(* IEC 61131-3 sources: RL_MAR/experiments/results/ablation/RL_MAR_DeepSeek-V3.2_full, 94 files *)

(* ---- hard_92.st ---- *)
TYPE
    BreakerState : STRUCT
        Opened : BOOL;
        Closed : BOOL;
    END_STRUCT;

    BreakerControl : STRUCT
        Trip : BOOL;
        Close : BOOL;
    END_STRUCT;

    BreakerData : STRUCT
        Control : BreakerControl;
        State : BreakerState;
    END_STRUCT;

    PointData : STRUCT
        Value : INT;
    END_STRUCT;
END_TYPE;

FUNCTION_BLOCK FB_BreakerControlSystem
VAR_INPUT
    B10_1_Trip : BOOL;
    B10_1_Close : BOOL;
    B10_2_Trip : BOOL;
    B10_2_Close : BOOL;
    B10_12_Trip : BOOL;
    B10_12_Close : BOOL;
    B54_Trip : BOOL;
    B54_Close : BOOL;
    B55_Trip : BOOL;
    B55_Close : BOOL;
    B56_Trip : BOOL;
    B56_Close : BOOL;
    B57_Trip : BOOL;
    B57_Close : BOOL;
END_VAR

VAR_OUTPUT
    Point_1a : INT;
    Point_2a : INT;
    Point_3a : INT;
    Point_4a : INT;
    B10_1_Opened : BOOL;
    B10_1_Closed : BOOL;
    B10_2_Opened : BOOL;
    B10_2_Closed : BOOL;
    B10_12_Opened : BOOL;
    B10_12_Closed : BOOL;
    B54_Opened : BOOL;
    B54_Closed : BOOL;
    B55_Opened : BOOL;
    B55_Closed : BOOL;
    B56_Opened : BOOL;
    B56_Closed : BOOL;
    B57_Opened : BOOL;
    B57_Closed : BOOL;
END_VAR

VAR
    SEL86_OUT : INT;
    MOVE89_OUT : INT;
    SEL66_OUT : INT;
    MOVE69_OUT : INT;
    SEL96_OUT : INT;
    MOVE99_OUT : INT;
    SEL106_OUT : INT;
    MOVE109_OUT : INT;
END_VAR

(* Breaker State Management *)
IF B10_1_Close = TRUE THEN
    B10_1_Closed := TRUE;
    B10_1_Opened := FALSE;
ELSIF B10_1_Trip = TRUE THEN
    B10_1_Closed := FALSE;
    B10_1_Opened := TRUE;
END_IF;

IF B10_2_Close = TRUE THEN
    B10_2_Closed := TRUE;
    B10_2_Opened := FALSE;
ELSIF B10_2_Trip = TRUE THEN
    B10_2_Closed := FALSE;
    B10_2_Opened := TRUE;
END_IF;

IF B10_12_Close = TRUE THEN
    B10_12_Closed := TRUE;
    B10_12_Opened := FALSE;
ELSIF B10_12_Trip = TRUE THEN
    B10_12_Closed := FALSE;
    B10_12_Opened := TRUE;
END_IF;

IF B54_Close = TRUE THEN
    B54_Closed := TRUE;
    B54_Opened := FALSE;
ELSIF B54_Trip = TRUE THEN
    B54_Closed := FALSE;
    B54_Opened := TRUE;
END_IF;

IF B55_Close = TRUE THEN
    B55_Closed := TRUE;
    B55_Opened := FALSE;
ELSIF B55_Trip = TRUE THEN
    B55_Closed := FALSE;
    B55_Opened := TRUE;
END_IF;

IF B56_Close = TRUE THEN
    B56_Closed := TRUE;
    B56_Opened := FALSE;
ELSIF B56_Trip = TRUE THEN
    B56_Closed := FALSE;
    B56_Opened := TRUE;
END_IF;

IF B57_Close = TRUE THEN
    B57_Closed := TRUE;
    B57_Opened := FALSE;
ELSIF B57_Trip = TRUE THEN
    B57_Closed := FALSE;
    B57_Opened := TRUE;
END_IF;

(* Point Calculations *)
IF (B54_Closed = TRUE) AND (((B10_12_Closed = TRUE) AND (B10_1_Closed = TRUE)) OR (B10_2_Closed = TRUE)) THEN
    Point_1a := 0;
ELSE
    Point_1a := 138;
END_IF;

IF (B55_Closed = TRUE) AND (((B10_12_Closed = TRUE) AND (B10_1_Closed = TRUE)) OR (B10_2_Closed = TRUE)) THEN
    Point_2a := 0;
ELSE
    Point_2a := 138;
END_IF;

IF (B56_Closed = TRUE) AND (((B10_12_Closed = TRUE) AND (B10_2_Closed = TRUE)) OR (B10_1_Closed = TRUE)) THEN
    Point_3a := 0;
ELSE
    Point_3a := 138;
END_IF;

IF (B57_Closed = TRUE) AND (((B10_12_Closed = TRUE) AND (B10_2_Closed = TRUE)) OR (B10_1_Closed = TRUE)) THEN
    Point_4a := 0;
ELSE
    Point_4a := 138;
END_IF;

END_FUNCTION_BLOCK;

(* ---- hard_93.st ---- *)
FUNCTION_BLOCK FB_CircuitControl
VAR_INPUT
    Reset_All_CB : BOOL;
    Current_Fault_on_TRSF1 : INT;
    Current_Fault_on_66BUS1 : INT;
END_VAR

VAR_OUTPUT
    Short_Circuit_TRSF1 : BOOL;
    Short_Circuit_66BUS : BOOL;
    Open_CB1_66KV : BOOL;
    Open_CB2_66KV : BOOL;
    Open_CB_TRSF1 : BOOL;
    Open_CB2_22KV : BOOL;
END_VAR

VAR
    Threshold500 : INT := 500;
    Prev_Open_CB2_22KV : BOOL;
    Prev_Open_CB1_66KV : BOOL;
    Prev_Open_CB_TRSF1 : BOOL;
    Temp_Open_CB2_22KV : BOOL;
    Temp_Open_CB1_66KV : BOOL;
    Temp_Open_CB_TRSF1 : BOOL;
END_VAR

(* Short circuit detection *)
Short_Circuit_66BUS := Current_Fault_on_66BUS1 > Threshold500;
Short_Circuit_TRSF1 := Current_Fault_on_TRSF1 > Threshold500;

(* Set Open_CB2_66KV to TRUE as specified *)
Open_CB2_66KV := TRUE;

(* Reset logic - when Reset_All_CB is TRUE, close all breakers and reset previous states *)
IF Reset_All_CB THEN
    Open_CB2_22KV := FALSE;
    Open_CB1_66KV := FALSE;
    Open_CB_TRSF1 := FALSE;
    Prev_Open_CB2_22KV := FALSE;
    Prev_Open_CB1_66KV := FALSE;
    Prev_Open_CB_TRSF1 := FALSE;
ELSE
    (* First calculation of breaker states *)
    Temp_Open_CB2_22KV := (NOT Prev_Open_CB2_22KV) AND ((Open_CB1_66KV AND Open_CB_TRSF1) OR Short_Circuit_66BUS);
    Temp_Open_CB1_66KV := (NOT Temp_Open_CB2_22KV) AND ((Prev_Open_CB1_66KV AND Open_CB_TRSF1) OR Short_Circuit_66BUS);
    Temp_Open_CB_TRSF1 := (NOT Temp_Open_CB2_22KV) AND ((Open_CB1_66KV AND Prev_Open_CB_TRSF1) OR Short_Circuit_66BUS);

    (* Update with Open_CB2_66KV and Short_Circuit_TRSF1 conditions *)
    Temp_Open_CB2_22KV := (NOT Prev_Open_CB2_22KV) AND ((Open_CB2_66KV AND Open_CB1_66KV AND Open_CB_TRSF1) OR Short_Circuit_TRSF1);
    Temp_Open_CB1_66KV := (NOT Temp_Open_CB2_22KV) AND ((Open_CB2_66KV AND Prev_Open_CB1_66KV AND Open_CB_TRSF1) OR Short_Circuit_TRSF1);
    Temp_Open_CB_TRSF1 := (NOT Temp_Open_CB2_22KV) AND ((Open_CB2_66KV AND Open_CB1_66KV AND Prev_Open_CB_TRSF1) OR Short_Circuit_TRSF1);

    (* Assign final values to outputs *)
    Open_CB2_22KV := Temp_Open_CB2_22KV;
    Open_CB1_66KV := Temp_Open_CB1_66KV;
    Open_CB_TRSF1 := Temp_Open_CB_TRSF1;

    (* Store current states as previous for next scan *)
    Prev_Open_CB2_22KV := Open_CB2_22KV;
    Prev_Open_CB1_66KV := Open_CB1_66KV;
    Prev_Open_CB_TRSF1 := Open_CB_TRSF1;
END_IF;

END_FUNCTION_BLOCK;

(* ---- hard_94.st ---- *)
FUNCTION_BLOCK FB_AdvancedCircuitBreakerControl
    VAR_INPUT
        S_AL1_P_B1 : BOOL;
        S_AL1_P_B2 : BOOL;
        S_AL1_MCB : BOOL;
        MCB_BUSY : BOOL;
        MCB_ERROR : BOOL;
        S_AL1_MCBR : BOOL;
        MCBR_BUSY : BOOL;
        MCBR_ERROR : BOOL;
        S_AL1_P_B3 : BOOL;
        S_AL1_MCB2 : BOOL;
        S_AL1_MCBR2 : BOOL;
    END_VAR

    VAR_OUTPUT
        E_AL1_B1 : BOOL;
        PUWS_AL1_B1_PLUS : BOOL;
        PUWS_AL1_B1_RIGHT : BOOL;
        PAS_AL1_PLUS : BOOL;
        PAS_AL1_TURN : BOOL;
    END_VAR

    VAR
        PPAL1 : BOOL := 1;
        PP0 : BOOL := 1;
        PP1 : BOOL := 0;
        PP2 : BOOL := 0;
        PP3 : BOOL := 0;
        PP4 : BOOL := 0;
        MCB : BOOL := 1;
        PP5 : BOOL := 0;
        PP7 : BOOL := 0;
        PPL3 : BOOL := 0;
        PPL4 : BOOL := 0;
        MCBR : BOOL := 1;
        PPL5 : BOOL := 0;
        PPL7 : BOOL := 0;
        STABLE : BOOL := 0;
        MCB_CONTROL : BOOL;
    END_VAR

    STABLE := 0;
    WHILE (STABLE = 0) DO
        STABLE := 1;
        IF PP0 AND (NOT MCB_CONTROL) AND (NOT PP1) THEN
            PP0 := 0;
            PP1 := 1;
            STABLE := 0;
        END_IF;
        IF PP1 AND S_AL1_P_B1 AND (NOT PP2) THEN
            PP1 := 0;
            PP2 := 1;
            STABLE := 0;
        END_IF;
        IF PP2 AND S_AL1_P_B2 AND (NOT MCB_CONTROL) AND (NOT PP3) THEN
            PP2 := 0;
            PP3 := 1;
            STABLE := 0;
        END_IF;
        IF PP3 AND S_AL1_MCB AND (NOT PP4) AND (NOT PP1) THEN
            PP3 := 0;
            PP4 := 1;
            PP1 := 1;
            STABLE := 0;
        END_IF;
        IF PP4 AND MCB AND MCB_BUSY AND (NOT PP5) THEN
            PP4 := 0;
            MCB := 0;
            PP5 := 1;
            STABLE := 0;
        END_IF;
        IF PP5 AND S_AL1_MCB2 AND (NOT PP7) AND (NOT MCB) THEN
            PP5 := 0;
            PP7 := 1;
            MCB := 1;
            STABLE := 0;
        END_IF;
        IF PP7 AND S_AL1_P_B3 THEN
            PP7 := 0;
            STABLE := 0;
        END_IF;
        IF PP2 AND S_AL1_P_B2 AND MCB_CONTROL AND (NOT PPL3) AND (NOT PP1) THEN
            PP2 := 0;
            PPL3 := 1;
            PP1 := 1;
            STABLE := 0;
        END_IF;
        IF PPL3 AND S_AL1_MCBR AND (NOT PPL4) THEN
            PPL3 := 0;
            PPL4 := 1;
            STABLE := 0;
        END_IF;
        IF PPL4 AND MCBR AND MCBR_BUSY AND (NOT PPL5) THEN
            PPL4 := 0;
            MCBR := 0;
            PPL5 := 1;
            STABLE := 0;
        END_IF;
        IF PPL5 AND S_AL1_MCBR2 AND (NOT PPL7) AND (NOT MCBR) THEN
            PPL5 := 0;
            PPL7 := 1;
            MCBR := 1;
            STABLE := 0;
        END_IF;
        IF PPL7 AND S_AL1_P_B3 THEN
            PPL7 := 0;
            STABLE := 0;
        END_IF;
    END_WHILE;

    IF PP0 OR PP1 THEN
        E_AL1_B1 := 1;
    END_IF;
    IF PP3 THEN
        MCB_CONTROL := 1;
    END_IF;
    IF PPL3 OR PPL4 THEN
        PAS_AL1_PLUS := 1;
        PAS_AL1_TURN := 1;
    END_IF;
    IF PPAL1 OR PP2 THEN
        PUWS_AL1_B1_PLUS := 1;
    END_IF;
    IF PP2 OR PP3 OR PPL3 THEN
        E_AL1_B1 := 0;
    END_IF;
    IF PP0 OR PP3 THEN
        MCB_CONTROL := 0;
    END_IF;
    IF PP0 OR PP3 OR PP4 THEN
        PAS_AL1_PLUS := 0;
        PAS_AL1_TURN := 0;
    END_IF;
    IF PPAL1 OR PP2 THEN
        PUWS_AL1_B1_RIGHT := 0;
    END_IF;
END_FUNCTION_BLOCK;

(* ---- hf_1.st ---- *)
FUNCTION_BLOCK StackMin
VAR_INPUT
    push : BOOL;
    pop : BOOL;
    reset : BOOL;
END_VAR

VAR_OUTPUT
    error : BOOL;
    status : WORD;
END_VAR

VAR_IN_OUT
    item : INT;
    stack : ARRAY[0..3] OF INT;
END_VAR

VAR
    top : INT := -1;
    i : INT;
    j : INT;
    minIndex : INT;
    minValue : INT;
END_VAR

IF reset THEN
    top := -1;
    error := FALSE;
    status := 16#0000;
ELSIF push THEN
    IF top >= 3 THEN
        error := TRUE;
        status := 16#8A04;
    ELSE
        top := top + 1;
        stack[top] := item;
        error := FALSE;
        status := 16#0000;
    END_IF;
ELSIF pop THEN
    IF top < 0 THEN
        error := TRUE;
        status := 16#8A05;
    ELSE
        minIndex := 0;
        minValue := stack[0];
        i := 1;
        WHILE i <= top DO
            IF stack[i] < minValue THEN
                minValue := stack[i];
                minIndex := i;
            END_IF;
            i := i + 1;
        END_WHILE;
        item := minValue;
        j := minIndex;
        WHILE j < top DO
            stack[j] := stack[j + 1];
            j := j + 1;
        END_WHILE;
        top := top - 1;
        error := FALSE;
        status := 16#0000;
    END_IF;
ELSE
    error := FALSE;
    status := 16#0000;
END_IF;

END_FUNCTION_BLOCK;

(* ---- hf_10.st ---- *)
FUNCTION_BLOCK FloatingAverage
VAR_INPUT
    cyclicExecution : BOOL;
    trigger : BOOL;
    value : REAL;
    windowSize : INT;
    reset : BOOL;
END_VAR

VAR_OUTPUT
    average : REAL;
    windowSizeReached : BOOL;
    error : BOOL;
    status : WORD;
END_VAR

VAR
    dataBuffer : ARRAY[1..100] OF REAL;
    bufferIndex : INT := 1;
    sum : REAL := 0.0;
    elementCount : INT := 0;
    triggerPrev : BOOL := FALSE;
    i : INT;
END_VAR

IF reset THEN
    sum := 0.0;
    average := 0.0;
    elementCount := 0;
    bufferIndex := 1;
    windowSizeReached := FALSE;
    error := FALSE;
    status := 16#0000;

    FOR i := 1 TO 100 DO
        dataBuffer[i] := 0.0;
    END_FOR;
ELSE
    IF (windowSize < 1) OR (windowSize > 100) THEN
        error := TRUE;
        status := 16#8200;
        average := 0.0;
        windowSizeReached := FALSE;
    ELSE
        error := FALSE;
        status := 16#0000;

        IF cyclicExecution THEN
            sum := sum - dataBuffer[bufferIndex];
            dataBuffer[bufferIndex] := value;
            sum := sum + value;

            bufferIndex := bufferIndex + 1;
            IF bufferIndex > windowSize THEN
                bufferIndex := 1;
            END_IF;

            IF elementCount < windowSize THEN
                elementCount := elementCount + 1;
            END_IF;
        ELSE
            IF trigger AND NOT triggerPrev THEN
                sum := sum - dataBuffer[bufferIndex];
                dataBuffer[bufferIndex] := value;
                sum := sum + value;

                bufferIndex := bufferIndex + 1;
                IF bufferIndex > windowSize THEN
                    bufferIndex := 1;
                END_IF;

                IF elementCount < windowSize THEN
                    elementCount := elementCount + 1;
                END_IF;
            END_IF;
            triggerPrev := trigger;
        END_IF;

        IF elementCount >= windowSize THEN
            windowSizeReached := TRUE;
            average := sum / INT_TO_REAL(windowSize);
        ELSE
            windowSizeReached := FALSE;
            IF elementCount > 0 THEN
                average := sum / INT_TO_REAL(elementCount);
            ELSE
                average := 0.0;
            END_IF;
        END_IF;
    END_IF;
END_IF;
END_FUNCTION_BLOCK

(* ---- hf_11.st ---- *)
FUNCTION_BLOCK FB_BottleProcessing
VAR_INPUT
    bottleSensor : BOOL;
    cleaningConfirmButton : BOOL;
    fillingConfirmButton : BOOL;
    cappingConfirmButton : BOOL;
    packingConfirmButton : BOOL;
    finishedButton : BOOL;
END_VAR

VAR_OUTPUT
    Pump_Motor : BOOL;
    Filling_Valve : BOOL;
    Capping_Machine : BOOL;
    Packing_Machine : BOOL;
    Completion_Light : BOOL;
END_VAR

VAR
    State : INT := 0;
END_VAR

CASE State OF
    0:
        Pump_Motor := FALSE;
        Filling_Valve := FALSE;
        Capping_Machine := FALSE;
        Packing_Machine := FALSE;
        Completion_Light := FALSE;

        IF bottleSensor THEN
            State := 1;
        END_IF;

    1:
        Pump_Motor := TRUE;
        Filling_Valve := FALSE;
        Capping_Machine := FALSE;
        Packing_Machine := FALSE;
        Completion_Light := FALSE;

        IF cleaningConfirmButton THEN
            State := 2;
        END_IF;

    2:
        Pump_Motor := FALSE;
        Filling_Valve := TRUE;
        Capping_Machine := FALSE;
        Packing_Machine := FALSE;
        Completion_Light := FALSE;

        IF fillingConfirmButton THEN
            State := 3;
        END_IF;

    3:
        Pump_Motor := FALSE;
        Filling_Valve := FALSE;
        Capping_Machine := TRUE;
        Packing_Machine := FALSE;
        Completion_Light := FALSE;

        IF cappingConfirmButton THEN
            State := 4;
        END_IF;

    4:
        Pump_Motor := FALSE;
        Filling_Valve := FALSE;
        Capping_Machine := FALSE;
        Packing_Machine := TRUE;
        Completion_Light := FALSE;

        IF packingConfirmButton THEN
            State := 5;
        END_IF;

    5:
        Pump_Motor := FALSE;
        Filling_Valve := FALSE;
        Capping_Machine := FALSE;
        Packing_Machine := FALSE;
        Completion_Light := TRUE;

        IF finishedButton THEN
            State := 0;
        END_IF;

    ELSE
        State := 0;
        Pump_Motor := FALSE;
        Filling_Valve := FALSE;
        Capping_Machine := FALSE;
        Packing_Machine := FALSE;
        Completion_Light := FALSE;
END_CASE;
END_FUNCTION_BLOCK

(* ---- hf_12.st ---- *)
FUNCTION_BLOCK MaterialMixing
VAR_INPUT
    estop : BOOL; (* Emergency Stop Signal, FALSE: Emergency stop triggered, TRUE: No emergency stop triggered *)
    opeMode : BOOL; (* Operation Mode, FALSE: Manual Operation Mode, TRUE: Automatic Operation Mode *)
    valveAStart : BOOL; (* Valve A Start Button *)
    valveBStart : BOOL; (* Valve B Start Button *)
    valveCStart : BOOL; (* Valve C Start Button *)
    valveDStart : BOOL; (* Valve D Start Button *)
    mixMotorStart : BOOL; (* Mixing Motor Start Button *)
    autoStart : BOOL; (* Automatic Start Button *)
    processMode : BOOL; (* Process Mode *)
    levelSensor : INT; (* Liquid Level Sensor, unit cm *)
    mixMotorComplete : BOOL; (* Mixing Complete Signal *)
END_VAR

VAR_OUTPUT
    valveARun : BOOL; (* Valve A Run Command *)
    valveBRun : BOOL; (* Valve B Run Command *)
    valveCRun : BOOL; (* Valve C Run Command *)
    valveDRun : BOOL; (* Valve D Run Command *)
    mixMotorRun : BOOL; (* Mixing Motor Run Command *)
END_VAR

VAR
    previousValveAStart : BOOL := FALSE;
    previousValveBStart : BOOL := FALSE;
    previousValveCStart : BOOL := FALSE;
    previousValveDStart : BOOL := FALSE;
    previousMixMotorStart : BOOL := FALSE;
    previousAutoStart : BOOL := FALSE;
END_VAR

(* Emergency Stop has highest priority - override all other logic *)
IF NOT estop THEN
    (* Automatic Operation Mode *)
    IF opeMode THEN
        (* Rising edge detection for autoStart button *)
        IF autoStart AND NOT previousAutoStart THEN
            valveARun := TRUE;
            valveBRun := FALSE;
            valveCRun := FALSE;
            valveDRun := FALSE;
            mixMotorRun := FALSE;
        END_IF;

        (* Automatic sequence logic *)
        IF valveARun AND (levelSensor >= 50) THEN
            valveARun := FALSE;
            valveBRun := TRUE;
        END_IF;

        IF valveBRun AND (levelSensor >= 80) THEN
            valveBRun := FALSE;
            IF processMode THEN
                valveCRun := TRUE;
            ELSE
                mixMotorRun := TRUE;
            END_IF;
        END_IF;

        IF valveCRun AND (levelSensor >= 100) THEN
            valveCRun := FALSE;
            mixMotorRun := TRUE;
        END_IF;

        IF mixMotorRun AND mixMotorComplete THEN
            mixMotorRun := FALSE;
            valveDRun := TRUE;
        END_IF;
    (* Manual Operation Mode *)
    ELSE
        (* Toggle logic with rising edge detection for manual buttons *)
        IF valveAStart AND NOT previousValveAStart THEN
            valveARun := NOT valveARun;
        END_IF;

        IF valveBStart AND NOT previousValveBStart THEN
            valveBRun := NOT valveBRun;
        END_IF;

        IF valveCStart AND NOT previousValveCStart THEN
            valveCRun := NOT valveCRun;
        END_IF;

        IF valveDStart AND NOT previousValveDStart THEN
            valveDRun := NOT valveDRun;
        END_IF;

        IF mixMotorStart AND NOT previousMixMotorStart THEN
            mixMotorRun := NOT mixMotorRun;
        END_IF;
    END_IF;
(* Emergency Stop active - force all outputs to FALSE *)
ELSE
    valveARun := FALSE;
    valveBRun := FALSE;
    valveCRun := FALSE;
    valveDRun := FALSE;
    mixMotorRun := FALSE;
END_IF;

(* Update previous state variables for edge detection *)
previousValveAStart := valveAStart;
previousValveBStart := valveBStart;
previousValveCStart := valveCStart;
previousValveDStart := valveDStart;
previousMixMotorStart := mixMotorStart;
previousAutoStart := autoStart;

END_FUNCTION_BLOCK;

(* ---- hf_13.st ---- *)
FUNCTION_BLOCK TON
VAR_INPUT
    IN : BOOL;
    PT : DINT;
    CYCLE_TIME : DINT;
END_VAR
VAR_OUTPUT
    Q : BOOL;
    ET : DINT;
END_VAR
VAR
    elapsedTimeInternal : DINT := 0;
    IN_PREV : BOOL := FALSE;
END_VAR

IF IN THEN
    IF NOT IN_PREV THEN
        elapsedTimeInternal := 0;
    END_IF;

    IF elapsedTimeInternal < PT THEN
        elapsedTimeInternal := elapsedTimeInternal + CYCLE_TIME;
        Q := FALSE;
    ELSE
        elapsedTimeInternal := PT;
        Q := TRUE;
    END_IF;

    ET := elapsedTimeInternal;
ELSE
    Q := FALSE;
    ET := 0;
    elapsedTimeInternal := 0;
END_IF;

IN_PREV := IN;
END_FUNCTION_BLOCK;

FUNCTION_BLOCK LightsControl
VAR_INPUT
    button1 : BOOL;
    button2 : BOOL;
    button3 : BOOL;
    CYCLE_TIME : DINT;
END_VAR
VAR_OUTPUT
    greenLight : BOOL;
    redLight : BOOL;
    yellowLight : BOOL;
END_VAR
VAR
    timerAuto : TON;
    timerGreen : TON;
    timerRed : TON;
    timerYellow : TON;
    currentState : INT := 0;
    autoRunTimer : BOOL;
END_VAR

IF NOT button1 THEN
    timerGreen(IN:=FALSE, PT:=1000, CYCLE_TIME:=CYCLE_TIME);
    timerRed(IN:=FALSE, PT:=1000, CYCLE_TIME:=CYCLE_TIME);
    timerYellow(IN:=FALSE, PT:=500, CYCLE_TIME:=CYCLE_TIME);

    IF NOT button2 AND NOT button3 THEN
        greenLight := FALSE;
        redLight := FALSE;
        yellowLight := FALSE;
    ELSIF button2 AND NOT button3 THEN
        greenLight := TRUE;
        timerRed(IN:=TRUE, PT:=1000, CYCLE_TIME:=CYCLE_TIME);
        redLight := timerRed.Q;
        yellowLight := FALSE;
    ELSIF NOT button2 AND button3 THEN
        redLight := TRUE;
        timerYellow(IN:=TRUE, PT:=500, CYCLE_TIME:=CYCLE_TIME);
        yellowLight := NOT timerYellow.Q;
        greenLight := FALSE;
    ELSIF button2 AND button3 THEN
        yellowLight := TRUE;
        timerGreen(IN:=TRUE, PT:=500, CYCLE_TIME:=CYCLE_TIME);
        greenLight := NOT timerGreen.Q;
        redLight := FALSE;
    END_IF;
ELSE
    autoRunTimer := TRUE;
    timerAuto(IN:=autoRunTimer, PT:=1000, CYCLE_TIME:=CYCLE_TIME);

    IF timerAuto.Q THEN
        currentState := currentState + 1;
        IF currentState > 2 THEN
            currentState := 0;
        END_IF;
        timerAuto(IN:=FALSE, PT:=1000, CYCLE_TIME:=CYCLE_TIME);
        timerAuto(IN:=TRUE, PT:=1000, CYCLE_TIME:=CYCLE_TIME);
    END_IF;

    CASE currentState OF
        0:
            greenLight := TRUE;
            redLight := FALSE;
            yellowLight := FALSE;
        1:
            greenLight := FALSE;
            redLight := TRUE;
            yellowLight := FALSE;
        2:
            greenLight := FALSE;
            redLight := FALSE;
            yellowLight := TRUE;
        ELSE
            currentState := 0;
            greenLight := TRUE;
            redLight := FALSE;
            yellowLight := FALSE;
    END_CASE;
END_IF;
END_FUNCTION_BLOCK;

(* ---- hf_14.st ---- *)
FUNCTION_BLOCK TruckGarage
VAR_INPUT
    enter_flag : BOOL;
    exit_flag : BOOL;
    VehicleNumber_in : INT;
END_VAR
VAR_OUTPUT
    truck_row : INT;
    truck_col : INT;
    truck_VehicleNumber : INT;
END_VAR
VAR_IN_OUT
    garage : ARRAY[1..3, 1..5] OF STRUCT
        Occupied : BOOL;
        VehicleNumber : INT;
    END_STRUCT;
END_VAR
VAR
    i : INT;
    j : INT;
    entry_found : BOOL;
    exit_found : BOOL;
END_VAR

// Initialize output
truck_row := 0;
truck_col := 0;
truck_VehicleNumber := 0;

// Entry logic
IF enter_flag THEN
    entry_found := FALSE;

    // Search from last row to first, last column to first
    FOR i := 3 TO 1 BY -1 DO
        FOR j := 5 TO 1 BY -1 DO
            IF NOT garage[i, j].Occupied AND NOT entry_found THEN
                // Allocate this space
                garage[i, j].Occupied := TRUE;
                garage[i, j].VehicleNumber := VehicleNumber_in;
                entry_found := TRUE;
            END_IF;
        END_FOR;
    END_FOR;
END_IF;

// Exit logic
IF exit_flag THEN
    exit_found := FALSE;

    // Search from first row to last, first column to last
    FOR i := 1 TO 3 DO
        FOR j := 1 TO 5 DO
            IF garage[i, j].Occupied AND (garage[i, j].VehicleNumber = VehicleNumber_in) AND NOT exit_found THEN
                // Release this space
                garage[i, j].Occupied := FALSE;
                garage[i, j].VehicleNumber := 0;

                // Set output information
                truck_row := i;
                truck_col := j;
                truck_VehicleNumber := VehicleNumber_in;
                exit_found := TRUE;
            END_IF;
        END_FOR;
    END_FOR;
END_IF;

END_FUNCTION_BLOCK

(* ---- hf_15.st ---- *)
FUNCTION_BLOCK FB_MergeBytes
VAR_INPUT
    byteArray : ARRAY[1..20] OF DINT; (* Byte array to be merged *)
END_VAR

VAR_OUTPUT
    dwordArray : ARRAY[1..10] OF DINT; (* Merged double word array *)
    mergeDwordNum : DINT; (* Actual number of merged double words *)
END_VAR

VAR
    i : DINT; (* Input byte index *)
    j : DINT; (* Byte counter within group (0-3) *)
    k : DINT; (* Output array index *)
    tempDword : DINT; (* Temporary storage for building double word *)
    currentByteValue : DINT; (* Temporary storage for current byte *)
END_VAR

VAR CONSTANT
    BYTE_ARRAY_SIZE : DINT := 20; (* Size of the input byte array *)
    DWORD_ARRAY_SIZE : DINT := 10; (* Size of the output DINT array *)
END_VAR

(* Initialize output count *)
mergeDwordNum := 0;

(* Clear output array *)
FOR k := 1 TO DWORD_ARRAY_SIZE DO
    dwordArray[k] := 0;
END_FOR;

(* Main merging loop *)
i := 1;
WHILE i <= BYTE_ARRAY_SIZE DO
    tempDword := 0;
    j := 0;

    (* Collect up to 4 bytes *)
    WHILE (j < 4) AND ((i + j) <= BYTE_ARRAY_SIZE) DO
        currentByteValue := byteArray[i + j];
        currentByteValue := currentByteValue AND 16#FF; (* Mask to keep only LSB *)
        tempDword := tempDword OR SHL(currentByteValue, 8 * j); (* Shift and combine *)
        j := j + 1;
    END_WHILE;

    (* Check if we have a complete group of 4 bytes *)
    IF j = 4 THEN
        k := mergeDwordNum + 1;

        (* Check if output array has space *)
        IF k <= DWORD_ARRAY_SIZE THEN
            dwordArray[k] := tempDword;
            mergeDwordNum := k;
        ELSE
            EXIT; (* Output array full *)
        END_IF;
    ELSE
        EXIT; (* Incomplete byte group *)
    END_IF;

    i := i + 4; (* Move to next group *)
END_WHILE;

END_FUNCTION_BLOCK;

(* ---- hf_16.st ---- *)
FUNCTION_BLOCK FB_LinearizeValue
VAR_INPUT
    InputValue : REAL; // Floating point input, raw measurement value
END_VAR

VAR_OUTPUT
    LinearizedValue : REAL; // Converted linear value
    Error : BOOL; // Error status indicator
    Status : WORD; // Status code
END_VAR

VAR
    // Internal constants for the piecewise linear segments
    RANGE1_IN_MIN : REAL := 1200.0;
    RANGE1_IN_MAX : REAL := 3600.0;
    RANGE1_OUT_MIN : REAL := 150.0;
    RANGE1_OUT_MAX : REAL := 240.0;

    RANGE2_IN_MIN : REAL := 3600.0;
    RANGE2_IN_MAX : REAL := 4800.0;
    RANGE2_OUT_MIN : REAL := 240.0;
    RANGE2_OUT_MAX : REAL := 560.0;

    RANGE3_IN_MIN : REAL := 4800.0;
    RANGE3_IN_MAX : REAL := 7000.0;
    RANGE3_OUT_MIN : REAL := 560.0;
    RANGE3_OUT_MAX : REAL := 720.0;

    // Status codes
    STATUS_SUCCESS : WORD := 16#0000;
    STATUS_OUT_OF_RANGE : WORD := 16#8001;
END_VAR

// Main execution logic
IF InputValue < RANGE1_IN_MIN THEN
    // Below minimum range
    LinearizedValue := RANGE1_OUT_MIN;
    Error := TRUE;
    Status := STATUS_OUT_OF_RANGE;
ELSIF InputValue >= RANGE1_IN_MIN AND InputValue <= RANGE1_IN_MAX THEN
    // Range 1: 1200 to 3600
    LinearizedValue := RANGE1_OUT_MIN + (InputValue - RANGE1_IN_MIN) *
                      (RANGE1_OUT_MAX - RANGE1_OUT_MIN) /
                      (RANGE1_IN_MAX - RANGE1_IN_MIN);
    Error := FALSE;
    Status := STATUS_SUCCESS;
ELSIF InputValue > RANGE1_IN_MAX AND InputValue <= RANGE2_IN_MAX THEN
    // Range 2: 3600 to 4800
    LinearizedValue := RANGE2_OUT_MIN + (InputValue - RANGE2_IN_MIN) *
                      (RANGE2_OUT_MAX - RANGE2_OUT_MIN) /
                      (RANGE2_IN_MAX - RANGE2_IN_MIN);
    Error := FALSE;
    Status := STATUS_SUCCESS;
ELSIF InputValue > RANGE2_IN_MAX AND InputValue <= RANGE3_IN_MAX THEN
    // Range 3: 4800 to 7000
    LinearizedValue := RANGE3_OUT_MIN + (InputValue - RANGE3_IN_MIN) *
                      (RANGE3_OUT_MAX - RANGE3_OUT_MIN) /
                      (RANGE3_IN_MAX - RANGE3_IN_MIN);
    Error := FALSE;
    Status := STATUS_SUCCESS;
ELSE
    // Above maximum range
    LinearizedValue := RANGE3_OUT_MAX;
    Error := TRUE;
    Status := STATUS_OUT_OF_RANGE;
END_IF;

END_FUNCTION_BLOCK

(* ---- hf_17.st ---- *)
FUNCTION_BLOCK FB_WarehouseManagement
VAR_INPUT
    requestIn : BOOL := FALSE;
    requestOut : BOOL := FALSE;
END_VAR

VAR_OUTPUT
    productNum : INT := 0;
    libFreeNum : INT := 9;
    error : BOOL := FALSE;
    status : WORD := 16#0000;
END_VAR

VAR_IN_OUT
    library : ARRAY[1..9] OF BOOL;
END_VAR

VAR
    i : INT;
    found : BOOL;
    initDone : BOOL := FALSE;
    errFull : WORD := 16#8001;
    errEmpty : WORD := 16#8002;
END_VAR

// Initialize library array on first execution
IF NOT initDone THEN
    i := 1;
    WHILE i <= 9 DO
        library[i] := FALSE;
        i := i + 1;
    END_WHILE;
    initDone := TRUE;
END_IF;

// Reset error status at start of each cycle
error := FALSE;
status := 16#0000;

// Handle storage request
IF requestIn THEN
    // Check if storage is full
    IF productNum >= 9 THEN
        error := TRUE;
        status := errFull;
    ELSE
        // Search for free position from highest to lowest index (9 to 1)
        found := FALSE;
        i := 9;
        WHILE i >= 1 AND NOT found DO
            IF NOT library[i] THEN
                library[i] := TRUE;
                productNum := productNum + 1;
                libFreeNum := libFreeNum - 1;
                found := TRUE;
            END_IF;
            i := i - 1;
        END_WHILE;

        // If no free position found despite productNum < 9, set error
        IF NOT found THEN
            error := TRUE;
            status := errFull;
        END_IF;
    END_IF;
END_IF;

// Handle retrieval request
IF requestOut THEN
    // Check if storage is empty
    IF productNum <= 0 THEN
        error := TRUE;
        status := errEmpty;
    ELSE
        // Search for occupied position from lowest to highest index (1 to 9)
        found := FALSE;
        i := 1;
        WHILE i <= 9 AND NOT found DO
            IF library[i] THEN
                library[i] := FALSE;
                productNum := productNum - 1;
                libFreeNum := libFreeNum + 1;
                found := TRUE;
            END_IF;
            i := i + 1;
        END_WHILE;

        // If no occupied position found despite productNum > 0, set error
        IF NOT found THEN
            error := TRUE;
            status := errEmpty;
        END_IF;
    END_IF;
END_IF;

END_FUNCTION_BLOCK

(* ---- hf_18.st ---- *)
FUNCTION_BLOCK FB_ColorLightControl
VAR_INPUT
    controlButton : BOOL;
END_VAR

VAR_OUTPUT
    greenLight : BOOL;
    redLight : BOOL;
    yellowLight : BOOL;
END_VAR

VAR
    state : INT := 1;
    lastControlButton : BOOL := FALSE;
END_VAR

IF controlButton AND NOT lastControlButton THEN
    CASE state OF
        1:
            greenLight := TRUE;
            redLight := FALSE;
            yellowLight := FALSE;
            state := 2;
        2:
            greenLight := FALSE;
            redLight := TRUE;
            yellowLight := FALSE;
            state := 3;
        3:
            greenLight := FALSE;
            redLight := FALSE;
            yellowLight := TRUE;
            state := 4;
        4:
            greenLight := TRUE;
            redLight := TRUE;
            yellowLight := TRUE;
            state := 5;
        5:
            greenLight := FALSE;
            redLight := FALSE;
            yellowLight := FALSE;
            state := 1;
        ELSE
            state := 1;
            greenLight := FALSE;
            redLight := FALSE;
            yellowLight := FALSE;
    END_CASE;
END_IF;

lastControlButton := controlButton;

END_FUNCTION_BLOCK;

(* ---- hf_19.st ---- *)
FUNCTION_BLOCK FB_DatabaseManager
    VAR_INPUT
        dataInput : ARRAY[0..5] OF BYTE;
        storeTrigger : BOOL;
        resetTrigger : BOOL;
    END_VAR

    VAR_OUTPUT
        usedSpace : INT := 0;
        remainingSpace : INT := 20;
        error : BOOL;
        status : WORD;
    END_VAR

    VAR_IN_OUT
        dataBase : ARRAY[1..20] OF BYTE;
    END_VAR

    VAR
        i : INT;
        dataLength : INT;
    END_VAR

    IF resetTrigger THEN
        FOR i := 1 TO 20 DO
            dataBase[i] := 0;
        END_FOR;
        usedSpace := 0;
        remainingSpace := 20;
        error := FALSE;
        status := 0;
    ELSIF storeTrigger THEN
        dataLength := dataInput[0];
        IF (dataLength <= 0) OR (dataLength > 5) THEN
            error := TRUE;
            status := 16#8001;
        ELSE
            IF (usedSpace + dataLength) > 20 THEN
                error := TRUE;
                status := 16#8002;
            ELSE
                FOR i := 1 TO dataLength DO
                    dataBase[usedSpace + i] := dataInput[i];
                END_FOR;
                usedSpace := usedSpace + dataLength;
                remainingSpace := 20 - usedSpace;
                error := FALSE;
                status := 0;
            END_IF;
        END_IF;
    END_IF;
END_FUNCTION_BLOCK;

(* ---- hf_2.st ---- *)
FUNCTION_BLOCK FindMinMaxValues
    VAR_INPUT
        values : ARRAY[1..10] OF DINT;
    END_VAR

    VAR_OUTPUT
        minValue : DINT;
        minValueIndex : DINT;
        maxValue : DINT;
        maxValueIndex : DINT;
    END_VAR

    VAR
        i : INT;
    END_VAR

    minValue := values[1];
    maxValue := values[1];
    minValueIndex := 1;
    maxValueIndex := 1;

    FOR i := 2 TO 10 DO
        IF values[i] < minValue THEN
            minValue := values[i];
            minValueIndex := i;
        END_IF;
        IF values[i] > maxValue THEN
            maxValue := values[i];
            maxValueIndex := i;
        END_IF;
    END_FOR;
END_FUNCTION_BLOCK;

(* ---- hf_20.st ---- *)
FUNCTION_BLOCK FB_ProductionLineControl
VAR_INPUT
    Mode : BOOL;
    ForwardButton : BOOL;
    ReverseButton : BOOL;
    SensorA : BOOL;
    SensorB : BOOL;
    SensorC : BOOL;
    ButtonA : BOOL;
    ButtonB : BOOL;
    ButtonC : BOOL;
END_VAR

VAR_OUTPUT
    MotorForward : BOOL;
    MotorReverse : BOOL;
    CompletionLight : BOOL;
END_VAR

VAR
    State : INT;
END_VAR

IF State = 0 THEN
    MotorForward := FALSE;
    MotorReverse := FALSE;
    CompletionLight := FALSE;
    State := 1;
END_IF;

IF NOT Mode THEN
    IF ForwardButton AND NOT ReverseButton THEN
        MotorForward := TRUE;
        MotorReverse := FALSE;
    ELSIF ReverseButton AND NOT ForwardButton THEN
        MotorForward := FALSE;
        MotorReverse := TRUE;
    ELSE
        MotorForward := FALSE;
        MotorReverse := FALSE;
    END_IF;
ELSE
    CASE State OF
        1:
            IF SensorA THEN
                State := 2;
            END_IF;
        2:
            IF ButtonA THEN
                MotorForward := TRUE;
                MotorReverse := FALSE;
                State := 3;
            END_IF;
        3:
            IF SensorB THEN
                MotorForward := FALSE;
                State := 4;
            END_IF;
        4:
            IF ButtonB THEN
                MotorForward := TRUE;
                MotorReverse := FALSE;
                State := 5;
            END_IF;
        5:
            IF SensorC THEN
                MotorForward := FALSE;
                State := 6;
            END_IF;
        6:
            IF ButtonC THEN
                CompletionLight := TRUE;
                State := 7;
            END_IF;
        7:
            IF NOT SensorC THEN
                CompletionLight := FALSE;
                State := 1;
            END_IF;
    END_CASE;
END_IF;

END_FUNCTION_BLOCK;

(* ---- hf_21.st ---- *)
FUNCTION_BLOCK FB_SplitNumber
VAR_INPUT
    InputNumber : INT;
END_VAR

VAR_OUTPUT
    Thousands : INT;
    Hundreds : INT;
    Tens : INT;
    Ones : INT;
    Min : INT;
    error : BOOL;
    status : WORD;
END_VAR

VAR
    tempNumber : INT;
    minValue : INT;
END_VAR

// Main logic
IF (InputNumber < 0) OR (InputNumber > 9999) THEN
    // Error condition
    error := TRUE;
    status := 16#8001;
    Thousands := 0;
    Hundreds := 0;
    Tens := 0;
    Ones := 0;
    Min := 0;
ELSE
    // Valid input - process normally
    error := FALSE;
    status := 0;

    // Digit separation
    Thousands := InputNumber / 1000;
    Hundreds := (InputNumber MOD 1000) / 100;
    Tens := (InputNumber MOD 100) / 10;
    Ones := InputNumber MOD 10;

    // Find minimum non-zero digit
    minValue := 32767;

    IF (Thousands <> 0) THEN
        minValue := minimal(minValue, Thousands);
    END_IF;

    IF (Hundreds <> 0) THEN
        minValue := minimal(minValue, Hundreds);
    END_IF;

    IF (Tens <> 0) THEN
        minValue := minimal(minValue, Tens);
    END_IF;

    IF (Ones <> 0) THEN
        minValue := minimal(minValue, Ones);
    END_IF;

    // Set Min output
    IF (minValue = 32767) THEN
        Min := 0;  // All digits were zero
    ELSE
        Min := minValue;
    END_IF;
END_IF;

END_FUNCTION_BLOCK

FUNCTION minimal : INT
VAR_INPUT
    IN1 : INT;
    IN2 : INT;
END_VAR

IF IN1 <= IN2 THEN
    minimal := IN1;
ELSE
    minimal := IN2;
END_IF;
END_FUNCTION

(* ---- hf_3.st ---- *)
FUNCTION_BLOCK MultiPumpCtrl
VAR_INPUT
    mode : BOOL;
    start : BOOL;
    stop : BOOL;
    priorities : ARRAY[1..5] OF INT;
    selections : ARRAY[1..5] OF BOOL;
END_VAR

VAR_OUTPUT
    RunComds : ARRAY[1..5] OF BOOL;
END_VAR

VAR
    i : INT;
    j : INT;
    maxPriority : INT;
    maxIndex : INT;
    runCount : INT;
    usedInAuto : ARRAY[1..5] OF BOOL;
END_VAR

IF stop THEN
    FOR i := 1 TO 5 DO
        RunComds[i] := FALSE;
    END_FOR;
ELSE
    IF start THEN
        IF NOT mode THEN
            FOR i := 1 TO 5 DO
                RunComds[i] := selections[i];
            END_FOR;
        ELSE
            FOR i := 1 TO 5 DO
                usedInAuto[i] := FALSE;
                RunComds[i] := FALSE;
            END_FOR;
            runCount := 0;
            WHILE runCount < 3 DO
                maxPriority := -32768;
                maxIndex := 0;
                FOR i := 1 TO 5 DO
                    IF (priorities[i] > maxPriority) AND NOT usedInAuto[i] THEN
                        maxPriority := priorities[i];
                        maxIndex := i;
                    END_IF;
                END_FOR;
                IF maxIndex > 0 THEN
                    usedInAuto[maxIndex] := TRUE;
                    RunComds[maxIndex] := TRUE;
                    runCount := runCount + 1;
                ELSE
                    EXIT;
                END_IF;
            END_WHILE;
        END_IF;
    ELSE
        FOR i := 1 TO 5 DO
            RunComds[i] := FALSE;
        END_FOR;
    END_IF;
END_IF;

END_FUNCTION_BLOCK;

(* ---- hf_4.st ---- *)
FUNCTION_BLOCK FB_CalculateDayOfYear
VAR_INPUT
    Year : INT;
    Month : INT;
    Day : INT;
END_VAR

VAR_OUTPUT
    DayOfYear : INT;
    error : BOOL;
    status : WORD;
END_VAR

VAR
    DaysInMonth : ARRAY[1..12] OF INT := [31, 28, 31, 30, 31, 30, 31, 31, 30, 31, 30, 31];
    i : INT;
    IsLeap : BOOL;
    MaxDay : INT;
END_VAR

DayOfYear := 0;
error := FALSE;
status := 0;

IF (Month < 1) OR (Month > 12) THEN
    error := TRUE;
    status := 16#8002;
    RETURN;
END_IF;

IsLeap := ((Year MOD 4) = 0) AND ((Year MOD 100) <> 0) OR ((Year MOD 400) = 0);
MaxDay := DaysInMonth[Month];

IF Month = 2 THEN
    IF IsLeap THEN
        MaxDay := 29;
    ELSE
        MaxDay := 28;
    END_IF;
END_IF;

IF (Day < 1) OR (Day > MaxDay) THEN
    error := TRUE;
    status := 16#8003;
    RETURN;
END_IF;

IF (Year < 1000) OR (Year > 3000) THEN
    error := TRUE;
    status := 16#8001;
    RETURN;
END_IF;

FOR i := 1 TO Month-1 DO
    DayOfYear := DayOfYear + DaysInMonth[i];
END_FOR;

DayOfYear := DayOfYear + Day;

IF IsLeap AND (Month > 2) THEN
    DayOfYear := DayOfYear + 1;
END_IF;

END_FUNCTION_BLOCK;

(* ---- hf_5.st ---- *)
FUNCTION_BLOCK SelectSort
VAR_INPUT
    exe : BOOL;
    seq : ARRAY[1..100] OF INT;
END_VAR

VAR_OUTPUT
    error : BOOL;
    status : WORD;
END_VAR

VAR
    i : INT;
    j : INT;
    min_idx : INT;
    temp : INT;
    n : INT;
    sort_successful : BOOL;
END_VAR

IF exe THEN
    error := FALSE;
    status := 16#0000;
    sort_successful := TRUE;

    n := 100;

    FOR i := 1 TO n-1 DO
        min_idx := i;

        FOR j := i+1 TO n DO
            IF seq[j] < seq[min_idx] THEN
                min_idx := j;
            END_IF;
        END_FOR;

        IF min_idx <> i THEN
            temp := seq[i];
            seq[i] := seq[min_idx];
            seq[min_idx] := temp;
        END_IF;
    END_FOR;

    IF NOT sort_successful THEN
        error := TRUE;
        status := 16#8A01;
    END_IF;

ELSE
    error := FALSE;
    status := 16#0000;
END_IF;

END_FUNCTION_BLOCK;

(* ---- hf_6.st ---- *)
FUNCTION_BLOCK RandomNumberGenerator
    VAR_INPUT
        minValue : DINT;
        maxValue : DINT;
        randomSeed_in : DINT;
    END_VAR

    VAR_OUTPUT
        error : BOOL;
        status : WORD;
        randomNumber : DINT;
    END_VAR

    VAR
        seed : DINT;
        range : DINT;
        offset : DINT;
    END_VAR

    IF minValue > maxValue THEN
        error := TRUE;
        status := 16#8200;
        randomNumber := 0;
        RETURN;
    END_IF;

    seed := randomSeed_in;
    IF seed < 0 THEN
        seed := seed * -1;
    END_IF;
    IF seed = 0 THEN
        seed := 1;
    END_IF;

    range := maxValue - minValue + 1;
    offset := seed MOD range;
    randomNumber := minValue + offset;

    error := FALSE;
    status := 16#0000;
END_FUNCTION_BLOCK;

(* ---- hf_7.st ---- *)
FUNCTION_BLOCK AnalogBatchConverter
    VAR_INPUT
        count : INT;
        analogValues : ARRAY[1..10] OF REAL;
    END_VAR

    VAR_OUTPUT
        channel_enable : ARRAY[1..10] OF BOOL;
        channel_hiLIM : ARRAY[1..10] OF REAL;
        channel_loLIM : ARRAY[1..10] OF REAL;
        channel_bipolar : ARRAY[1..10] OF BOOL;
        channel_measuringMode : ARRAY[1..10] OF INT;
        channel_retVal : ARRAY[1..10] OF WORD;
        channel_outputValue : ARRAY[1..10] OF REAL;
    END_VAR

    VAR
        i : INT;
        rawValue : REAL;
        scaleFactor : REAL;
    END_VAR

    FOR i := 1 TO 10 DO
        IF i <= count AND channel_enable[i] THEN
            channel_retVal[i] := 16#0000;
            rawValue := analogValues[i];

            CASE channel_measuringMode[i] OF
                0:
                    IF channel_hiLIM[i] <= channel_loLIM[i] THEN
                        channel_retVal[i] := 16#8002;
                        channel_outputValue[i] := 0.0;
                    ELSE
                        IF channel_bipolar[i] THEN
                            scaleFactor := (rawValue + 27648.0) / 55296.0;
                        ELSE
                            scaleFactor := rawValue / 27648.0;
                        END_IF;
                        channel_outputValue[i] := channel_loLIM[i] + scaleFactor * (channel_hiLIM[i] - channel_loLIM[i]);
                    END_IF;
                1:
                    channel_outputValue[i] := rawValue / 10.0;
                2:
                    channel_outputValue[i] := rawValue / 100.0;
                ELSE
                    channel_retVal[i] := 16#8001;
                    channel_outputValue[i] := 0.0;
            END_CASE;
        ELSE
            channel_outputValue[i] := 0.0;
            channel_retVal[i] := 16#0000;
        END_IF;
    END_FOR;
END_FUNCTION_BLOCK;

(* ---- hf_8.st ---- *)
FUNCTION_BLOCK FB_HexDigitAnalyzer
VAR_INPUT
    InputNumber : INT;
END_VAR

VAR_OUTPUT
    Thousands : INT;
    Hundreds : INT;
    Tens : INT;
    Ones : INT;
    MinDigit : INT;
    error : BOOL;
    status : WORD;
END_VAR

VAR
    tempMin : INT;
    digit : INT;
END_VAR

METHOD ProcessDigits : BOOL
VAR_INPUT
END_VAR
VAR
END_VAR

    // Input validation
    IF (InputNumber < 0) OR (InputNumber > 9999) THEN
        error := TRUE;
        status := 16#8001;
        Thousands := 0;
        Hundreds := 0;
        Tens := 0;
        Ones := 0;
        MinDigit := 0;
        RETURN FALSE;
    ELSE
        error := FALSE;
        status := 16#0000;
    END_IF;

    // Digit separation
    Thousands := InputNumber / 1000;
    Hundreds := (InputNumber MOD 1000) / 100;
    Tens := (InputNumber MOD 100) / 10;
    Ones := InputNumber MOD 10;

    // Minimum non-zero digit detection
    tempMin := 32767; // Maximum INT value

    // Check Thousands
    digit := Thousands;
    IF digit > 0 THEN
        IF digit < tempMin THEN
            tempMin := digit;
        END_IF;
    END_IF;

    // Check Hundreds
    digit := Hundreds;
    IF digit > 0 THEN
        IF digit < tempMin THEN
            tempMin := digit;
        END_IF;
    END_IF;

    // Check Tens
    digit := Tens;
    IF digit > 0 THEN
        IF digit < tempMin THEN
            tempMin := digit;
        END_IF;
    END_IF;

    // Check Ones
    digit := Ones;
    IF digit > 0 THEN
        IF digit < tempMin THEN
            tempMin := digit;
        END_IF;
    END_IF;

    // Set MinDigit
    IF tempMin = 32767 THEN
        MinDigit := 0; // All digits were zero
    ELSE
        MinDigit := tempMin;
    END_IF;

    RETURN TRUE;
END_METHOD

// Main execution
ProcessDigits();

(* ---- hf_9.st ---- *)
FUNCTION_BLOCK ShellSortFB
    VAR_INPUT
        sortDirection : BOOL;
        arr : ARRAY[1..1000] OF DINT;
    END_VAR

    VAR_OUTPUT
        error : BOOL;
        status : WORD;
        sorted_arr : ARRAY[1..1000] OF DINT;
    END_VAR

    VAR
        gap : DINT;
        i : DINT;
        j : DINT;
        temp : DINT;
        n : DINT;
        continueLoop : BOOL;
    END_VAR

    n := 1000;
    error := FALSE;
    status := 16#0000;
    sorted_arr := arr;

    IF n <= 1 THEN
        error := TRUE;
        status := 16#8200;
        RETURN;
    END_IF;

    IF n > 1000 THEN
        error := TRUE;
        status := 16#8201;
        RETURN;
    END_IF;

    gap := n / 2;
    WHILE gap > 0 DO
        i := gap + 1;
        WHILE i <= n DO
            temp := sorted_arr[i];
            j := i;
            continueLoop := TRUE;
            WHILE (j > gap) AND continueLoop DO
                IF NOT sortDirection THEN
                    IF sorted_arr[j - gap] <= temp THEN
                        continueLoop := FALSE;
                    ELSE
                        sorted_arr[j] := sorted_arr[j - gap];
                        j := j - gap;
                    END_IF;
                ELSE
                    IF sorted_arr[j - gap] >= temp THEN
                        continueLoop := FALSE;
                    ELSE
                        sorted_arr[j] := sorted_arr[j - gap];
                        j := j - gap;
                    END_IF;
                END_IF;
            END_WHILE;
            sorted_arr[j] := temp;
            i := i + 1;
        END_WHILE;
        gap := gap / 2;
    END_WHILE;
END_FUNCTION_BLOCK;

(* ---- med_22.st ---- *)
FUNCTION_BLOCK CottonCandyMachine
VAR_INPUT
    SugarLevel : REAL; (* Input for sugar level *)
    SpinningSpeed : INT; (* Input for spinning speed *)
END_VAR

VAR_OUTPUT
    SugarFeeder : BOOL; (* Output to control sugar feeding *)
    MotorSpeed : INT; (* Output to control spinning motor speed *)
END_VAR

(* Main logic body begins here *)
IF SugarLevel < 10.0 THEN
    SugarFeeder := TRUE;
ELSE
    SugarFeeder := FALSE;
END_IF;

IF SpinningSpeed > 0 THEN
    MotorSpeed := SpinningSpeed;
ELSE
    MotorSpeed := 0;
END_IF;

END_FUNCTION_BLOCK;

(* ---- med_23.st ---- *)
FUNCTION_BLOCK SmartIrrigationSystem
VAR_INPUT
    SoilMoistureSensor1 : REAL;
    SoilMoistureSensor2 : REAL;
    WeatherForecast : INT; (* 0: Sunny, 1: Rainy, 2: Cloudy *)
END_VAR

VAR_OUTPUT
    WaterPump : BOOL;
END_VAR

VAR
    SoilMoistureThreshold : REAL := 30.0;
END_VAR

IF WeatherForecast = 1 THEN
    WaterPump := FALSE;
ELSIF WeatherForecast = 0 THEN
    IF (SoilMoistureSensor1 < SoilMoistureThreshold) OR (SoilMoistureSensor2 < SoilMoistureThreshold) THEN
        WaterPump := TRUE;
    ELSE
        WaterPump := FALSE;
    END_IF;
ELSE
    WaterPump := FALSE;
END_IF;

END_FUNCTION_BLOCK;

(* ---- med_24.st ---- *)
FUNCTION_BLOCK AutomaticDoorControl
VAR_INPUT
    ProximitySensor : BOOL;
    ElapsedTime : DINT;
END_VAR

VAR_OUTPUT
    DoorOpen : BOOL;
END_VAR

VAR
    DoorOpenDuration : DINT := 5000;
    CurrentState : INT := 0;
    NextState : INT := 0;
END_VAR

CASE CurrentState OF
    0:
        DoorOpen := FALSE;
        IF ProximitySensor THEN
            NextState := 1;
        ELSE
            NextState := 0;
        END_IF;
    1:
        DoorOpen := TRUE;
        NextState := 2;
    2:
        DoorOpen := TRUE;
        IF (NOT ProximitySensor) OR (ElapsedTime >= DoorOpenDuration) THEN
            NextState := 0;
        ELSE
            NextState := 2;
        END_IF;
    ELSE
        NextState := 0;
END_CASE;

CurrentState := NextState;

END_FUNCTION_BLOCK;

(* ---- med_25.st ---- *)
FUNCTION_BLOCK WastewaterControl
VAR_INPUT
    InFlow : REAL;
    OutFlow : REAL;
    pH : REAL;
    TankLvl : REAL;
END_VAR

VAR_OUTPUT
    Pump1 : BOOL;
    Pump2 : BOOL;
    Valve1 : BOOL;
    Valve2 : BOOL;
END_VAR

VAR
    LowInFlow : REAL := 100.0;
    HighOutFlow : REAL := 90.0;
    DesiredPH : REAL := 7.0;
    HighTankLvl : REAL := 80.0;
END_VAR

IF InFlow < LowInFlow THEN
    Pump1 := TRUE;
ELSE
    Pump1 := FALSE;
END_IF;

IF OutFlow > HighOutFlow THEN
    Pump2 := TRUE;
ELSE
    Pump2 := FALSE;
END_IF;

IF pH < DesiredPH THEN
    Valve1 := TRUE;
ELSE
    Valve1 := FALSE;
END_IF;

IF TankLvl > HighTankLvl THEN
    Valve2 := TRUE;
ELSE
    Valve2 := FALSE;
END_IF;

END_FUNCTION_BLOCK;

(* ---- med_26.st ---- *)
FUNCTION_BLOCK BookSorting
    VAR_INPUT
        RFID1 : BOOL;
        RFID2 : BOOL;
        RFID3 : BOOL;
    END_VAR

    VAR_OUTPUT
        Motor : BOOL;
        Bin1 : BOOL;
        Bin2 : BOOL;
        Bin3 : BOOL;
    END_VAR

    VAR
        (* No internal variables needed for this simple logic *)
    END_VAR

    (* Main logic body *)
    Motor := RFID1 OR RFID2 OR RFID3;

    IF RFID1 AND NOT RFID2 AND NOT RFID3 THEN
        Bin1 := TRUE;
        Bin2 := FALSE;
        Bin3 := FALSE;
    ELSIF RFID2 AND NOT RFID1 AND NOT RFID3 THEN
        Bin1 := FALSE;
        Bin2 := TRUE;
        Bin3 := FALSE;
    ELSIF RFID3 AND NOT RFID1 AND NOT RFID2 THEN
        Bin1 := FALSE;
        Bin2 := FALSE;
        Bin3 := TRUE;
    ELSE
        Bin1 := FALSE;
        Bin2 := FALSE;
        Bin3 := FALSE;
    END_IF;

END_FUNCTION_BLOCK;

(* ---- med_27.st ---- *)
FUNCTION_BLOCK FlowerArrangingMachine
VAR_INPUT
    FlowerTypeSensor : INT; (* Input for detecting flower type *)
    FlowerColorSensor : INT; (* Input for detecting flower color *)
END_VAR

VAR_OUTPUT
    ArrangingMechanism : INT; (* Output for controlling arranging mechanism *)
    ConveyorBelt : BOOL; (* Output for controlling conveyor belt *)
END_VAR

VAR
    (* No internal variables required for this combinational logic *)
END_VAR

(* Main logic body *)
IF (FlowerTypeSensor = 1) AND (FlowerColorSensor = 1) THEN
    ArrangingMechanism := 1;
ELSIF (FlowerTypeSensor = 1) AND (FlowerColorSensor = 2) THEN
    ArrangingMechanism := 2;
ELSIF (FlowerTypeSensor = 2) AND (FlowerColorSensor = 1) THEN
    ArrangingMechanism := 3;
ELSIF (FlowerTypeSensor = 2) AND (FlowerColorSensor = 2) THEN
    ArrangingMechanism := 4;
ELSE
    ArrangingMechanism := 0;
END_IF;

ConveyorBelt := ArrangingMechanism <> 0;

END_FUNCTION_BLOCK;

(* ---- med_28.st ---- *)
FUNCTION_BLOCK HomeBrewingSystem
VAR_INPUT
    TemperatureSensor : REAL; (* Input for temperature measurement *)
    WaterFlowSensor : REAL; (* Input for water flow measurement *)
    BrewingStartTime : TIME; (* Input for brewing start time *)
    BrewingDuration : TIME; (* Input for brewing duration *)
END_VAR

VAR_OUTPUT
    HeatingElement : BOOL; (* Output for heating element *)
    AgitationMotor : BOOL; (* Output for agitation motor *)
    HopsDispenser : BOOL; (* Output for hops dispenser *)
    FermentationTank : BOOL; (* Output for fermentation tank *)
END_VAR

VAR
    ElapsedTime : TIME;
END_VAR

(* Main logic body *)
ElapsedTime := BrewingDuration;

IF TemperatureSensor < 65.0 THEN
    HeatingElement := TRUE;
ELSE
    HeatingElement := FALSE;
END_IF;

IF WaterFlowSensor > 0.5 THEN
    AgitationMotor := TRUE;
ELSE
    AgitationMotor := FALSE;
END_IF;

IF ElapsedTime >= T#5h THEN
    HopsDispenser := TRUE;
ELSE
    HopsDispenser := FALSE;
END_IF;

IF ElapsedTime >= T#48h THEN
    FermentationTank := TRUE;
ELSE
    FermentationTank := FALSE;
END_IF;

END_FUNCTION_BLOCK;

(* ---- med_29.st ---- *)
FUNCTION_BLOCK DocumentFilingSystem
VAR_INPUT
    DocumentInlet : BOOL; (* Input to detect the arrival of a document *)
    CategorySelector : INT; (* Input to select the document category *)
END_VAR

VAR_OUTPUT
    ConveyorMotor : BOOL; (* Output to control the conveyor motor *)
    StorageBin1 : BOOL; (* Output to activate storage bin 1 *)
    StorageBin2 : BOOL; (* Output to activate storage bin 2 *)
    StorageBin3 : BOOL; (* Output to activate storage bin 3 *)
    StorageBin4 : BOOL; (* Output to activate storage bin 4 *)
END_VAR

VAR
    bValidCategory : BOOL;
END_VAR

(* Main logic body begins here *)

bValidCategory := (CategorySelector >= 1) AND (CategorySelector <= 4);

IF DocumentInlet AND bValidCategory THEN
    ConveyorMotor := TRUE;

    CASE CategorySelector OF
        1:
            StorageBin1 := TRUE;
            StorageBin2 := FALSE;
            StorageBin3 := FALSE;
            StorageBin4 := FALSE;
        2:
            StorageBin1 := FALSE;
            StorageBin2 := TRUE;
            StorageBin3 := FALSE;
            StorageBin4 := FALSE;
        3:
            StorageBin1 := FALSE;
            StorageBin2 := FALSE;
            StorageBin3 := TRUE;
            StorageBin4 := FALSE;
        4:
            StorageBin1 := FALSE;
            StorageBin2 := FALSE;
            StorageBin3 := FALSE;
            StorageBin4 := TRUE;
        ELSE
            StorageBin1 := FALSE;
            StorageBin2 := FALSE;
            StorageBin3 := FALSE;
            StorageBin4 := FALSE;
    END_CASE;
ELSE
    ConveyorMotor := FALSE;
    StorageBin1 := FALSE;
    StorageBin2 := FALSE;
    StorageBin3 := FALSE;
    StorageBin4 := FALSE;
END_IF;

END_FUNCTION_BLOCK;

(* ---- med_30.st ---- *)
FUNCTION_BLOCK MuseumClimateControl
VAR_INPUT
    HumiditySensor : REAL;
    TemperatureSensor : REAL;
    LightSensor : BOOL;
END_VAR

VAR_OUTPUT
    HVACSystem : BOOL;
    Humidifier : BOOL;
    Dehumidifier : BOOL;
    LightControl : BOOL;
END_VAR

VAR
    TargetHumidity : REAL := 50.0;
    TargetTemperature : REAL := 20.0;
    LightThreshold : BOOL := TRUE;
END_VAR

IF HumiditySensor < TargetHumidity THEN
    Humidifier := TRUE;
    Dehumidifier := FALSE;
ELSIF HumiditySensor > TargetHumidity THEN
    Humidifier := FALSE;
    Dehumidifier := TRUE;
ELSE
    Humidifier := FALSE;
    Dehumidifier := FALSE;
END_IF;

IF TemperatureSensor <> TargetTemperature THEN
    HVACSystem := TRUE;
ELSE
    HVACSystem := FALSE;
END_IF;

IF LightSensor AND LightThreshold THEN
    LightControl := FALSE;
ELSE
    LightControl := TRUE;
END_IF;

END_FUNCTION_BLOCK;

(* ---- med_31.st ---- *)
FUNCTION_BLOCK ChargingStationControl
VAR_INPUT
    EVConnected : BOOL;
    EVVoltage : REAL;
    EVCurrent : REAL;
    EVStateOfCharge : REAL;
    ChargingTimer : TIME;
END_VAR

VAR_OUTPUT
    EVCharging : BOOL;
END_VAR

VAR
    VoltageOK : BOOL;
    CurrentOK : BOOL;
    SOCNotFull : BOOL;
    TimerOK : BOOL;
END_VAR

    VoltageOK := EVVoltage > 350.0;
    CurrentOK := EVCurrent <= 32.0;
    SOCNotFull := EVStateOfCharge < 100.0;
    TimerOK := ChargingTimer <= T#2h;

    IF EVConnected AND VoltageOK AND CurrentOK AND SOCNotFull AND TimerOK THEN
        EVCharging := TRUE;
    ELSE
        EVCharging := FALSE;
    END_IF;

END_FUNCTION_BLOCK;

(* ---- med_32.st ---- *)
FUNCTION_BLOCK GreenhouseWateringSystem
    VAR_INPUT
        SoilMoistureSensor : REAL;   (* Input for soil moisture level (0-100%) *)
        ResponseDelay : TIME := T#5s;  (* Example response delay for the system *)
    END_VAR

    VAR_OUTPUT
        SprinklersOn : BOOL := FALSE;         (* Output for controlling sprinklers - on/off *)
    END_VAR

    VAR
        LastMoistureReading : REAL;
        DelayTimer : TON;
        DelayActive : BOOL;
    END_VAR

    (* Store the current moisture reading *)
    LastMoistureReading := SoilMoistureSensor;

    (* Timer logic for response delay *)
    DelayTimer(
        IN := DelayActive,
        PT := ResponseDelay
    );

    (* Main control logic with hysteresis and delay consideration *)
    IF NOT DelayTimer.Q THEN
        (* Timer not yet elapsed - maintain current state *)
        IF DelayActive THEN
            (* Delay in progress - keep sprinklers in their current state *)
            SprinklersOn := SprinklersOn;
        ELSE
            (* No delay active - evaluate moisture thresholds *)
            IF SoilMoistureSensor < 30.0 THEN
                IF NOT SprinklersOn THEN
                    DelayActive := TRUE;
                END_IF;
                SprinklersOn := TRUE;
            ELSIF SoilMoistureSensor > 70.0 THEN
                IF SprinklersOn THEN
                    DelayActive := TRUE;
                END_IF;
                SprinklersOn := FALSE;
            ELSE
                (* Between 30% and 70% - maintain current state *)
                SprinklersOn := SprinklersOn;
                DelayActive := FALSE;
            END_IF;
        END_IF;
    ELSE
        (* Timer has elapsed - reset delay flag *)
        DelayActive := FALSE;
        DelayTimer(IN := FALSE, PT := ResponseDelay);
    END_IF;

END_FUNCTION_BLOCK;

(* ---- med_33.st ---- *)
FUNCTION_BLOCK RoboticArmColorSorting
VAR_INPUT
    ColorSensorRed : BOOL;   (* Input: Red color sensor *)
    ColorSensorGreen : BOOL;  (* Input: Green color sensor *)
    ColorSensorBlue : BOOL;   (* Input: Blue color sensor *)
END_VAR

VAR_OUTPUT
    RoboticArmMove : BOOL := FALSE;     (* Output: Control for robotic arm movement *)
    BinRed : BOOL := FALSE;           (* Output: Activate red bin *)
    BinGreen : BOOL := FALSE;         (* Output: Activate green bin *)
    BinBlue : BOOL := FALSE;          (* Output: Activate blue bin *)
END_VAR

(* Main logic body begins here *)
IF ColorSensorRed OR ColorSensorGreen OR ColorSensorBlue THEN
    RoboticArmMove := TRUE;

    (* Priority-based bin activation to ensure only one bin is active at a time *)
    IF ColorSensorRed THEN
        BinRed := TRUE;
        BinGreen := FALSE;
        BinBlue := FALSE;
    ELSIF ColorSensorGreen THEN
        BinRed := FALSE;
        BinGreen := TRUE;
        BinBlue := FALSE;
    ELSIF ColorSensorBlue THEN
        BinRed := FALSE;
        BinGreen := FALSE;
        BinBlue := TRUE;
    ELSE
        BinRed := FALSE;
        BinGreen := FALSE;
        BinBlue := FALSE;
    END_IF;
ELSE
    RoboticArmMove := FALSE;
    BinRed := FALSE;
    BinGreen := FALSE;
    BinBlue := FALSE;
END_IF;
END_FUNCTION_BLOCK;

(* ---- med_34.st ---- *)
FUNCTION_BLOCK CoffeeMachineControl
VAR_INPUT
    StartButton : BOOL;
    ElapsedTime : DINT; (* Time elapsed since the start of the current process, in milliseconds *)
END_VAR

VAR_OUTPUT
    WaterHeating : BOOL;
    GrinderRunning : BOOL;
    Brewing : BOOL;
    WaterHeated : BOOL;
    GrinderFinished : BOOL;
    CoffeeReady : BOOL;
END_VAR

VAR
    CurrentState : INT := 0;
    ProcessStartTime : DINT := 0;
    WaterHeatingDuration : DINT := 30000;
    GrinderDuration : DINT := 15000;
    BrewingDuration : DINT := 60000;
    WaterHeatedFlag : BOOL := FALSE;
    GrinderFinishedFlag : BOOL := FALSE;
    CoffeeReadyFlag : BOOL := FALSE;
    ProcessActive : BOOL := FALSE;
END_VAR

(* State Definitions:
   0: Idle
   1: Water Heating
   2: Grinder Running
   3: Brewing
*)

(* Reset all outputs when StartButton is not pressed *)
IF NOT StartButton THEN
    CurrentState := 0;
    ProcessStartTime := 0;
    WaterHeating := FALSE;
    GrinderRunning := FALSE;
    Brewing := FALSE;
    WaterHeated := FALSE;
    GrinderFinished := FALSE;
    CoffeeReady := FALSE;
    WaterHeatedFlag := FALSE;
    GrinderFinishedFlag := FALSE;
    CoffeeReadyFlag := FALSE;
    ProcessActive := FALSE;
    RETURN;
END_IF;

(* Main state machine *)
CASE CurrentState OF
    0: (* Idle - Start water heating when button pressed and water not heated *)
        IF StartButton AND NOT WaterHeatedFlag THEN
            CurrentState := 1;
            ProcessStartTime := ElapsedTime;
            WaterHeating := TRUE;
            ProcessActive := TRUE;
        END_IF;

    1: (* Water Heating *)
        IF (ElapsedTime - ProcessStartTime) >= WaterHeatingDuration THEN
            WaterHeating := FALSE;
            WaterHeatedFlag := TRUE;
            WaterHeated := TRUE;
            CurrentState := 2;
            ProcessStartTime := ElapsedTime;
            GrinderRunning := TRUE;
        END_IF;

    2: (* Grinder Running *)
        IF (ElapsedTime - ProcessStartTime) >= GrinderDuration THEN
            GrinderRunning := FALSE;
            GrinderFinishedFlag := TRUE;
            GrinderFinished := TRUE;
            CurrentState := 3;
            ProcessStartTime := ElapsedTime;
            Brewing := TRUE;
        END_IF;

    3: (* Brewing *)
        IF (ElapsedTime - ProcessStartTime) >= BrewingDuration THEN
            Brewing := FALSE;
            CoffeeReadyFlag := TRUE;
            CoffeeReady := TRUE;
            CurrentState := 0;
            ProcessActive := FALSE;
        END_IF;

    ELSE
        CurrentState := 0;
END_CASE;

END_FUNCTION_BLOCK;

(* ---- med_35.st ---- *)
FUNCTION_BLOCK FB_SimpleCalculation
VAR_INPUT
    INPUT_VAR1 : INT := 2;
    VAR2 : INT := 0;
END_VAR

VAR_OUTPUT
    OUTPUT_VAR1 : INT;
    OUTPUT_VAR2 : INT;
END_VAR

VAR
    i : INT;
    COUNTER2 : INT := 0;
END_VAR

// Initialization
OUTPUT_VAR1 := INPUT_VAR1;
OUTPUT_VAR2 := VAR2;
COUNTER2 := 0;

// Loop 1: Multiply OUTPUT_VAR1 by 2, five times
FOR i := 1 TO 5 DO
    OUTPUT_VAR1 := OUTPUT_VAR1 * 2;
END_FOR;

// Loop 2: Increment OUTPUT_VAR2 five times
WHILE COUNTER2 < 5 DO
    OUTPUT_VAR2 := OUTPUT_VAR2 + 1;
    COUNTER2 := COUNTER2 + 1;
END_WHILE;

END_FUNCTION_BLOCK;

(* ---- med_36.st ---- *)
FUNCTION_BLOCK FB_ExpandedPoint
    VAR_INPUT
        INPUT_VAR2 : INT;
        INPUT_VAR1_X : INT;
        INPUT_VAR1_Y : INT;
        INPUT_VAR3_X : INT := 1;
        INPUT_VAR3_Y : INT := 2;
    END_VAR

    VAR_OUTPUT
        OUTPUT_VAR2 : INT;
        OUTPUT_VAR1_X : INT;
        OUTPUT_VAR1_Y : INT;
        OUTPUT_VAR3_X : INT;
        OUTPUT_VAR3_Y : INT;
    END_VAR

    OUTPUT_VAR2 := INPUT_VAR2;
    OUTPUT_VAR1_X := 1;
    OUTPUT_VAR1_Y := 2;
    OUTPUT_VAR3_X := 100;
    OUTPUT_VAR3_Y := -7000;
END_FUNCTION_BLOCK

(* ---- med_37.st ---- *)
FUNCTION_BLOCK FB_RealValueAdjuster
VAR_INPUT
    x_in : REAL;
END_VAR

VAR_OUTPUT
    x_out : REAL;
END_VAR

VAR
    x : REAL;
END_VAR

x := x_in;

IF x_in = 0.0 THEN
    x := x + 1.0;
END_IF;

IF x_in <> 0.0 THEN
    x := x + 1.0;
END_IF;

IF REAL_TO_INT(x_in) <> 0 THEN
    x := x + 1.0;
END_IF;

x_out := x;
END_FUNCTION_BLOCK;

(* ---- med_38.st ---- *)
FUNCTION_BLOCK SolarPanelTracking
VAR_INPUT
    SolarIntensity : REAL;      (* Input: Solar intensity in percentage *)
    CurrentTime : TIME;         (* Input: Current time of day *)
END_VAR

VAR_OUTPUT
    PanelAngle : REAL := 0.0;   (* Output: Panel angle in degrees *)
END_VAR

VAR
    SunriseTime : TIME := T#6H;    (* Sunrise time set to 6 AM *)
    SunsetTime : TIME := T#18H;    (* Sunset time set to 6 PM *)
    NoonTime : TIME := T#12H;      (* Noon time set to 12 PM *)
    MorningAngle : REAL := 30.0;   (* Angle during morning *)
    NoonAngle : REAL := 60.0;      (* Angle during noon *)
    EveningAngle : REAL := 30.0;   (* Angle during evening *)
    State : INT := 0;              (* State variable for state machine *)
END_VAR

(* Main state machine logic *)
CASE State OF
    0: (* INIT *)
        PanelAngle := 0.0;
        State := 1;

    1: (* CHECK_TIME *)
        IF (CurrentTime < SunriseTime) OR (CurrentTime >= SunsetTime) THEN
            State := 2;
        ELSIF (CurrentTime < NoonTime) THEN
            State := 3;
        ELSE
            State := 4;
        END_IF;

    2: (* NIGHTTIME *)
        PanelAngle := 0.0;
        State := 1;

    3: (* MORNING *)
        PanelAngle := MorningAngle;
        IF (SolarIntensity >= 90.0) THEN
            State := 5;
        ELSE
            State := 1;
        END_IF;

    4: (* AFTERNOON_EVENING *)
        PanelAngle := EveningAngle;
        IF (SolarIntensity >= 90.0) THEN
            State := 5;
        ELSE
            State := 1;
        END_IF;

    5: (* HIGH_INTENSITY *)
        PanelAngle := NoonAngle;
        State := 1;

    ELSE
        State := 0;
END_CASE;

(* Apply boundary limits to ensure angle stays within 0-90 degrees *)
IF PanelAngle < 0.0 THEN
    PanelAngle := 0.0;
ELSIF PanelAngle > 90.0 THEN
    PanelAngle := 90.0;
END_IF;

END_FUNCTION_BLOCK;

(* ---- med_39.st ---- *)
FUNCTION_BLOCK WindTurbineControl
VAR_INPUT
    WindSpeedSensor : REAL; (* Input for measuring wind speed *)
    GeneratorSpeedSensor : REAL; (* Input for measuring generator speed *)
END_VAR

VAR_OUTPUT
    BladePitch : INT; (* Output for blade pitch control (degrees) *)
    GeneratorSpeed : REAL; (* Output for generator speed control (RPM) *)
END_VAR

(* Main logic body begins here *)
IF WindSpeedSensor <= 3.0 THEN
    BladePitch := -5;
    GeneratorSpeed := 500.0;
ELSIF (WindSpeedSensor > 3.0) AND (WindSpeedSensor <= 5.0) THEN
    BladePitch := 0;
    GeneratorSpeed := 800.0;
ELSIF WindSpeedSensor > 5.0 THEN
    BladePitch := 5;
    GeneratorSpeed := 1000.0;
END_IF;

END_FUNCTION_BLOCK

(* ---- med_40.st ---- *)
FUNCTION_BLOCK RockClimbingWallControl
VAR_INPUT
    UserWeightSensor : REAL; (* Input for measuring the user's weight *)
    WallDifficultyLevel : INT; (* Input for setting the wall's initial difficulty level *)
    WallHeight : REAL; (* Input for setting the wall's height *)
    RouteSelector : INT; (* Input for selecting a climbing route *)
END_VAR

VAR_OUTPUT
    ClimbingMotorSpeed : REAL; (* Output for controlling the climbing wall motor speed *)
    WallLights : BOOL; (* Output for controlling wall lighting *)
END_VAR

VAR
    (* No internal variables required for basic logic *)
END_VAR

(* Main logic body *)
IF UserWeightSensor > 60.0 THEN
    ClimbingMotorSpeed := 1.0;
ELSE
    ClimbingMotorSpeed := 0.8;
END_IF;

CASE RouteSelector OF
    1: WallDifficultyLevel := 1;
    2: WallDifficultyLevel := 2;
    3: WallDifficultyLevel := 3;
    ELSE
        WallDifficultyLevel := 0;
END_CASE;

IF WallHeight > 5.0 THEN
    WallLights := TRUE;
ELSE
    WallLights := FALSE;
END_IF;

END_FUNCTION_BLOCK;

(* ---- med_41.st ---- *)
FUNCTION_BLOCK FishTankControl
VAR_INPUT
    OxygenLevel : REAL; (* Input for oxygen level in the tank *)
    WaterTemperature : REAL; (* Input for water temperature *)
    FeedingTime : TIME; (* Time for scheduled feeding *)
    CurrentTime : TIME; (* Current system time *)
END_VAR

VAR_OUTPUT
    OxygenValve : BOOL; (* Output to control oxygen supply *)
    Heater : BOOL; (* Output to control the heater *)
    Feeder : BOOL; (* Output to control the fish feeder *)
END_VAR

(* Main logic body begins here *)
IF OxygenLevel < 5.0 THEN
    OxygenValve := TRUE;
ELSE
    OxygenValve := FALSE;
END_IF;

IF WaterTemperature < 25.0 THEN
    Heater := TRUE;
ELSE
    Heater := FALSE;
END_IF;

IF CurrentTime >= FeedingTime THEN
    Feeder := TRUE;
ELSE
    Feeder := FALSE;
END_IF;

END_FUNCTION_BLOCK;

(* ---- med_42.st ---- *)
FUNCTION_BLOCK RetractableRoofControl
    VAR_INPUT
        RainSensor : BOOL; (* Input to detect rain *)
        WindSensor : BOOL; (* Input to detect wind *)
        TemperatureSensor : REAL; (* Input to measure temperature *)
    END_VAR

    VAR_OUTPUT
        RoofMotor : BOOL; (* Output to control the roof motor *)
    END_VAR

    VAR
        (* No internal variables needed for this simple logic *)
    END_VAR

    (* Main logic body begins here *)
    IF RainSensor AND WindSensor THEN
        RoofMotor := FALSE;
    ELSIF RainSensor AND NOT WindSensor THEN
        RoofMotor := TRUE;
    ELSIF NOT RainSensor AND TemperatureSensor < 20.0 THEN
        RoofMotor := TRUE;
    ELSIF NOT RainSensor AND TemperatureSensor >= 20.0 THEN
        RoofMotor := FALSE;
    END_IF;

END_FUNCTION_BLOCK;

(* ---- med_43.st ---- *)
FUNCTION_BLOCK SandwichMaker
VAR_INPUT
    BreadFeeder : BOOL; (* Input: Detects the presence of bread slices *)
    Ingredient1 : BOOL; (* Input: Detects the presence of Ingredient 1 (e.g., cheese) *)
    Ingredient2 : BOOL; (* Input: Detects the presence of Ingredient 2 (e.g., lettuce) *)
    Ingredient3 : BOOL; (* Input: Detects the presence of Ingredient 3 (e.g., tomatoes) *)
    Condiment1 : BOOL; (* Input: Detects the presence of Condiment 1 (e.g., mayo) *)
    Condiment2 : BOOL; (* Input: Detects the presence of Condiment 2 (e.g., mustard) *)
END_VAR

VAR_OUTPUT
    ConveyorMotor : BOOL; (* Output: Controls the conveyor belt motor *)
    AssembleMotor : BOOL; (* Output: Controls the sandwich assembly motor *)
END_VAR

VAR
    SliceCount : INT := 0; (* Counter for bread slices *)
    BreadFeederPrev : BOOL := FALSE; (* Previous state for edge detection *)
    AllIngredientsPresent : BOOL; (* Helper variable for condition *)
END_VAR

(* Edge detection for bread slice counting *)
IF BreadFeeder AND NOT BreadFeederPrev THEN
    SliceCount := SliceCount + 1;
END_IF;
BreadFeederPrev := BreadFeeder;

(* Conveyor motor control *)
ConveyorMotor := BreadFeeder;

(* Check if all ingredients and condiments are present *)
AllIngredientsPresent := Ingredient1 AND Ingredient2 AND Ingredient3 AND Condiment1 AND Condiment2;

(* Assembly motor control with reset condition *)
IF (SliceCount >= 2) AND AllIngredientsPresent THEN
    AssembleMotor := TRUE;
    SliceCount := 0; (* Reset counter after assembly *)
ELSE
    AssembleMotor := FALSE;
END_IF;

END_FUNCTION_BLOCK;

(* ---- med_44.st ---- *)
FUNCTION_BLOCK DroneChargingStation
VAR_INPUT
    Drone1BatteryLevel : INT := 0; (* Battery level of Drone 1 (0-100%) *)
    Drone2BatteryLevel : INT := 0; (* Battery level of Drone 2 (0-100%) *)
    Drone3BatteryLevel : INT := 0; (* Battery level of Drone 3 (0-100%) *)
    ChargingTime : TIME := T#30s; (* Charging time required for each drone *)
END_VAR

VAR_OUTPUT
    Drone1Status : BOOL := FALSE; (* Status of Drone 1 *)
    Drone2Status : BOOL := FALSE; (* Status of Drone 2 *)
    Drone3Status : BOOL := FALSE; (* Status of Drone 3 *)
    ChargingStationStatus : BOOL := FALSE; (* Charging station status *)
    DroneDeployed : BOOL := FALSE; (* Indicates if a drone is deployed *)
END_VAR

VAR
    TimeRemaining : TIME := T#0s; (* Remaining charging time for the current charging operation *)
    CurrentState : INT := 0; (* 0=IDLE, 1=CHARGING_DRONE1, 2=CHARGING_DRONE2, 3=CHARGING_DRONE3 *)
    NextState : INT := 0; (* Next state for state machine *)
    RecallCondition : BOOL := FALSE; (* Battery < 10% recall condition *)
END_VAR

(* Main state machine logic *)
RecallCondition := (Drone1BatteryLevel < 10) OR (Drone2BatteryLevel < 10) OR (Drone3BatteryLevel < 10);

CASE CurrentState OF
    0: (* IDLE STATE *)
        (* Reset all drone charging statuses *)
        Drone1Status := FALSE;
        Drone2Status := FALSE;
        Drone3Status := FALSE;
        ChargingStationStatus := FALSE;

        (* Check for deployment recall condition *)
        IF DroneDeployed AND RecallCondition THEN
            DroneDeployed := FALSE;
        END_IF;

        (* Determine next state *)
        IF NOT DroneDeployed THEN
            (* Check for drones needing charging in priority order *)
            IF Drone1BatteryLevel < 20 THEN
                NextState := 1;  (* Start charging Drone 1 *)
                TimeRemaining := ChargingTime;
            ELSIF Drone2BatteryLevel < 20 THEN
                NextState := 2;  (* Start charging Drone 2 *)
                TimeRemaining := ChargingTime;
            ELSIF Drone3BatteryLevel < 20 THEN
                NextState := 3;  (* Start charging Drone 3 *)
                TimeRemaining := ChargingTime;
            ELSE
                NextState := 0;  (* Stay in IDLE *)
            END_IF;
        ELSE
            NextState := 0;  (* Stay in IDLE if drone is deployed *)
        END_IF;

    1: (* CHARGING_DRONE1 STATE *)
        (* Set charging status for Drone 1 only *)
        Drone1Status := TRUE;
        Drone2Status := FALSE;
        Drone3Status := FALSE;
        ChargingStationStatus := TRUE;

        (* Decrement charging timer *)
        IF TimeRemaining > T#0s THEN
            TimeRemaining := TimeRemaining - T#1ms;
        END_IF;

        (* Determine next state *)
        IF TimeRemaining <= T#0s THEN
            NextState := 0;  (* Return to IDLE when charging complete *)
        ELSIF DroneDeployed AND RecallCondition THEN
            DroneDeployed := FALSE;
            NextState := 0;  (* Return to IDLE for recall *)
        ELSE
            NextState := 1;  (* Continue charging *)
        END_IF;

    2: (* CHARGING_DRONE2 STATE *)
        (* Set charging status for Drone 2 only *)
        Drone1Status := FALSE;
        Drone2Status := TRUE;
        Drone3Status := FALSE;
        ChargingStationStatus := TRUE;

        (* Decrement charging timer *)
        IF TimeRemaining > T#0s THEN
            TimeRemaining := TimeRemaining - T#1ms;
        END_IF;

        (* Determine next state *)
        IF TimeRemaining <= T#0s THEN
            NextState := 0;  (* Return to IDLE when charging complete *)
        ELSIF DroneDeployed AND RecallCondition THEN
            DroneDeployed := FALSE;
            NextState := 0;  (* Return to IDLE for recall *)
        ELSE
            NextState := 2;  (* Continue charging *)
        END_IF;

    3: (* CHARGING_DRONE3 STATE *)
        (* Set charging status for Drone 3 only *)
        Drone1Status := FALSE;
        Drone2Status := FALSE;
        Drone3Status := TRUE;
        ChargingStationStatus := TRUE;

        (* Decrement charging timer *)
        IF TimeRemaining > T#0s THEN
            TimeRemaining := TimeRemaining - T#1ms;
        END_IF;

        (* Determine next state *)
        IF TimeRemaining <= T#0s THEN
            NextState := 0;  (* Return to IDLE when charging complete *)
        ELSIF DroneDeployed AND RecallCondition THEN
            DroneDeployed := FALSE;
            NextState := 0;  (* Return to IDLE for recall *)
        ELSE
            NextState := 3;  (* Continue charging *)
        END_IF;

    ELSE
        (* Default case - return to IDLE *)
        NextState := 0;
END_CASE;

(* Update current state for next cycle *)
CurrentState := NextState;

END_FUNCTION_BLOCK;

(* ---- med_45.st ---- *)
FUNCTION_BLOCK AutomatedSmoothieMaker
    VAR_INPUT
        BananaAvailable : BOOL;
        BerryMixAvailable : BOOL;
        SpinachAvailable : BOOL;
        YogurtAvailable : BOOL;
        CustomerPreference : INT;
    END_VAR

    VAR_OUTPUT
        BlenderMotor : BOOL;
        Dispenser : BOOL;
    END_VAR

    VAR
        RecipeValid : BOOL;
        IngredientsAvailable : BOOL;
    END_VAR

    RecipeValid := FALSE;
    IngredientsAvailable := FALSE;

    CASE CustomerPreference OF
        1:
            IF BananaAvailable AND BerryMixAvailable AND YogurtAvailable THEN
                RecipeValid := TRUE;
                IngredientsAvailable := TRUE;
            END_IF;
        2:
            IF BerryMixAvailable AND SpinachAvailable AND YogurtAvailable THEN
                RecipeValid := TRUE;
                IngredientsAvailable := TRUE;
            END_IF;
        3:
            IF BananaAvailable AND SpinachAvailable AND YogurtAvailable THEN
                RecipeValid := TRUE;
                IngredientsAvailable := TRUE;
            END_IF;
        ELSE
            RecipeValid := FALSE;
            IngredientsAvailable := FALSE;
    END_CASE;

    IF RecipeValid AND IngredientsAvailable THEN
        BlenderMotor := TRUE;
        Dispenser := TRUE;
    ELSE
        BlenderMotor := FALSE;
        Dispenser := FALSE;
    END_IF;
END_FUNCTION_BLOCK;

(* ---- med_46.st ---- *)
FUNCTION_BLOCK PrecisionEngravingMachine
VAR_INPUT
    DesignSelection : INT;
END_VAR

VAR_OUTPUT
    EngravingDepth : REAL;
    EngravingSpeed : REAL;
    ZAxisMotor : BOOL;
    EngravingMotor : BOOL;
END_VAR

VAR
    CalculatedDepth : REAL;
    CalculatedSpeed : REAL;
END_VAR

CASE DesignSelection OF
    1:
        CalculatedDepth := 0.1;
        CalculatedSpeed := 10.0;
        ZAxisMotor := TRUE;
        EngravingMotor := TRUE;
    2:
        CalculatedDepth := 0.2;
        CalculatedSpeed := 8.0;
        ZAxisMotor := TRUE;
        EngravingMotor := TRUE;
    3:
        CalculatedDepth := 0.15;
        CalculatedSpeed := 12.0;
        ZAxisMotor := TRUE;
        EngravingMotor := TRUE;
    ELSE
        CalculatedDepth := 0.0;
        CalculatedSpeed := 0.0;
        ZAxisMotor := FALSE;
        EngravingMotor := FALSE;
END_CASE;

EngravingDepth := CalculatedDepth;
EngravingSpeed := CalculatedSpeed;

END_FUNCTION_BLOCK;

(* ---- med_47.st ---- *)
FUNCTION_BLOCK WindowCleaningSystem
    VAR_INPUT
        StartButton : BOOL;
        EmergencyStop : BOOL;
        UpperLimit : BOOL;
        LowerLimit : BOOL;
    END_VAR

    VAR_OUTPUT
        ElevatorUp : BOOL;
        ElevatorDown : BOOL;
        RotateClockwise : BOOL;
        WaterPump : BOOL;
    END_VAR

    VAR
        CleaningInProgress : BOOL;
        StartButtonPrev : BOOL;
        StartRisingEdge : BOOL;
    END_VAR

    (* Emergency Stop has highest priority - force safe state *)
    IF EmergencyStop THEN
        CleaningInProgress := FALSE;
        ElevatorUp := FALSE;
        ElevatorDown := FALSE;
        RotateClockwise := FALSE;
        WaterPump := FALSE;
        StartButtonPrev := FALSE;
    ELSE
        (* Detect rising edge of StartButton *)
        StartRisingEdge := StartButton AND NOT StartButtonPrev;
        StartButtonPrev := StartButton;

        (* Start sequence only on rising edge when idle and at lower limit *)
        IF NOT CleaningInProgress AND StartRisingEdge AND LowerLimit THEN
            CleaningInProgress := TRUE;
        END_IF;

        (* Main operational logic *)
        IF CleaningInProgress THEN
            (* Ascent phase: move up until upper limit is reached *)
            IF NOT UpperLimit THEN
                ElevatorUp := TRUE;
                ElevatorDown := FALSE;
                RotateClockwise := FALSE;
                WaterPump := FALSE;
            (* Descent and cleaning phase: move down with tools active until lower limit *)
            ELSE
                ElevatorUp := FALSE;
                ElevatorDown := TRUE;
                RotateClockwise := TRUE;
                WaterPump := TRUE;
            END_IF;

            (* End of cycle: reached lower limit *)
            IF LowerLimit THEN
                CleaningInProgress := FALSE;
                ElevatorDown := FALSE;
                RotateClockwise := FALSE;
                WaterPump := FALSE;
            END_IF;
        ELSE
            (* Idle state: all outputs off *)
            ElevatorUp := FALSE;
            ElevatorDown := FALSE;
            RotateClockwise := FALSE;
            WaterPump := FALSE;
        END_IF;
    END_IF;
END_FUNCTION_BLOCK;

(* ---- med_48.st ---- *)
FUNCTION_BLOCK ChargingStationControl
VAR_INPUT
    EVConnected : BOOL;
    EVVoltage : REAL;
    EVCurrent : REAL;
    EVStateOfCharge : REAL;
    ChargingTimer : TIME;
    MinimumVoltage : REAL;
    MaximumCurrent : REAL;
    MinimumSOC : REAL;
    ChargingVoltage : REAL;
    ChargingCurrent : REAL;
    MaximumChargingTime : TIME;
END_VAR

VAR_OUTPUT
    EVCharging : BOOL;
END_VAR

VAR
    bStartConditionsMet : BOOL;
    bStopConditionActive : BOOL;
END_VAR

    (* Evaluate all start conditions simultaneously *)
    bStartConditionsMet := EVConnected
        AND (EVVoltage > MinimumVoltage)
        AND (EVCurrent <= MaximumCurrent)
        AND (EVStateOfCharge < 100.0)
        AND (ChargingTimer <= MaximumChargingTime);

    (* Evaluate stop conditions - any single condition stops charging *)
    bStopConditionActive := NOT EVConnected
        OR (EVVoltage <= MinimumVoltage)
        OR (EVCurrent > MaximumCurrent)
        OR (EVStateOfCharge >= 100.0)
        OR (ChargingTimer > MaximumChargingTime);

    (* Final charging decision: start conditions met AND no stop conditions active *)
    EVCharging := bStartConditionsMet AND NOT bStopConditionActive;

END_FUNCTION_BLOCK;

(* ---- med_49.st ---- *)
FUNCTION_BLOCK SmartHVACSystem
VAR_INPUT
    TemperatureSensor : REAL; (* Temperature sensor reading *)
    HumiditySensor : REAL; (* Humidity sensor reading *)
END_VAR

VAR_OUTPUT
    HVACMode : INT := 0; (* HVAC operating mode: 0=Off, 1=Cooling, 2=Heating, 3=Ventilation *)
    HVACFanSpeed : INT := 0; (* Fan speed: 0=Off, 1=Low, 2=Medium, 3=High *)
END_VAR

VAR
    DesiredTemperature : REAL := 24.0; (* Desired temperature setting *)
    DesiredHumidity : REAL := 50.0; (* Desired humidity setting *)
    TemperatureThreshold : REAL := 1.0; (* Temperature tolerance threshold *)
    HumidityThreshold : REAL := 5.0; (* Humidity tolerance threshold *)
    AdjustedHumidity : REAL; (* Sanitized humidity input *)
    AdjustedTemperature : REAL; (* Sanitized temperature input *)
    NeedsVentilation : BOOL; (* Flag for ventilation requirement *)
    NeedsHeating : BOOL; (* Flag for heating requirement *)
    NeedsCooling : BOOL; (* Flag for cooling requirement *)
END_VAR

    (* Input Sanitization *)
    IF HumiditySensor < 0.0 THEN
        AdjustedHumidity := 0.0;
    ELSIF HumiditySensor > 100.0 THEN
        AdjustedHumidity := 100.0;
    ELSE
        AdjustedHumidity := HumiditySensor;
    END_IF;

    IF TemperatureSensor < -50.0 THEN
        AdjustedTemperature := -50.0;
    ELSIF TemperatureSensor > 100.0 THEN
        AdjustedTemperature := 100.0;
    ELSE
        AdjustedTemperature := TemperatureSensor;
    END_IF;

    (* Determine System Requirements *)
    NeedsVentilation := AdjustedHumidity < (DesiredHumidity - HumidityThreshold);
    NeedsHeating := AdjustedTemperature < (DesiredTemperature - TemperatureThreshold);
    NeedsCooling := AdjustedTemperature > (DesiredTemperature + TemperatureThreshold);

    (* Control Logic with Prioritization *)
    IF NeedsHeating THEN
        HVACMode := 2;
        HVACFanSpeed := 3;
    ELSIF NeedsCooling THEN
        HVACMode := 1;
        HVACFanSpeed := 3;
    ELSIF NeedsVentilation THEN
        HVACMode := 3;
        HVACFanSpeed := 3;
    ELSE
        HVACMode := 0;
        HVACFanSpeed := 0;
    END_IF;

END_FUNCTION_BLOCK;

(* ---- med_50.st ---- *)
FUNCTION_BLOCK CarParkingSystem
VAR_INPUT
    NewCarSlot : INT; (* Input for new car arrival slot number *)
END_VAR

VAR_OUTPUT
    Elevator1Busy : BOOL; (* Elevator 1 status - busy or idle *)
    Elevator2Busy : BOOL; (* Elevator 2 status - busy or idle *)
    Elevator1Position : INT; (* Elevator 1 current position *)
    Elevator2Position : INT; (* Elevator 2 current position *)
END_VAR

VAR
    Elevator1Target : INT; (* Elevator 1 target floor *)
    Elevator2Target : INT; (* Elevator 2 target floor *)
    CarSlots : ARRAY[1..100] OF BOOL; (* Array to represent parking slots - TRUE if occupied *)
    CurrentSlot : INT; (* Loop counter for scanning slots *)
END_VAR

(* Process new car arrival *)
IF (NewCarSlot >= 1) AND (NewCarSlot <= 100) THEN
    IF NOT CarSlots[NewCarSlot] THEN
        IF NewCarSlot <= 50 THEN
            IF NOT Elevator1Busy THEN
                Elevator1Target := NewCarSlot;
                Elevator1Busy := TRUE;
            END_IF;
        ELSE
            IF NOT Elevator2Busy THEN
                Elevator2Target := NewCarSlot;
                Elevator2Busy := TRUE;
            END_IF;
        END_IF;
        CarSlots[NewCarSlot] := TRUE;
    END_IF;
END_IF;

(* Elevator 1 motion control *)
IF Elevator1Busy THEN
    IF Elevator1Position < Elevator1Target THEN
        Elevator1Position := Elevator1Position + 1;
    ELSIF Elevator1Position > Elevator1Target THEN
        Elevator1Position := Elevator1Position - 1;
    ELSE
        Elevator1Busy := FALSE;
    END_IF;
ELSE
    (* Idle: scan for new tasks in assigned range (slots 1-50) *)
    FOR CurrentSlot := 1 TO 50 DO
        IF CarSlots[CurrentSlot] THEN
            Elevator1Target := CurrentSlot;
            Elevator1Busy := TRUE;
            EXIT;
        END_IF;
    END_FOR;
END_IF;

(* Elevator 2 motion control *)
IF Elevator2Busy THEN
    IF Elevator2Position < Elevator2Target THEN
        Elevator2Position := Elevator2Position + 1;
    ELSIF Elevator2Position > Elevator2Target THEN
        Elevator2Position := Elevator2Position - 1;
    ELSE
        Elevator2Busy := FALSE;
    END_IF;
ELSE
    (* Idle: scan for new tasks in assigned range (slots 51-100) *)
    FOR CurrentSlot := 51 TO 100 DO
        IF CarSlots[CurrentSlot] THEN
            Elevator2Target := CurrentSlot;
            Elevator2Busy := TRUE;
            EXIT;
        END_IF;
    END_FOR;
END_IF;

END_FUNCTION_BLOCK;

(* ---- med_51.st ---- *)
FUNCTION_BLOCK PizzaMakingMachine
VAR_INPUT
    StartButton : BOOL;
    StopButton : BOOL;
    DoughReadySensor : BOOL;
    ToppingsReadySensor : BOOL;
    BakingDoneSensor : BOOL;
END_VAR

VAR_OUTPUT
    DoughRollerMotor : BOOL;
    ToppingDispenser : BOOL;
    ConveyorMotor : BOOL;
    OvenHeater : BOOL;
    OvenTemperature : INT;
END_VAR

VAR
    SystemActive : BOOL;
    BakingActive : BOOL;
END_VAR

(* Emergency stop handling - highest priority *)
IF StopButton THEN
    SystemActive := FALSE;
    BakingActive := FALSE;
    DoughRollerMotor := FALSE;
    ToppingDispenser := FALSE;
    ConveyorMotor := FALSE;
    OvenHeater := FALSE;
    OvenTemperature := 0;
    RETURN;
END_IF;

(* System activation *)
IF StartButton AND NOT SystemActive THEN
    SystemActive := TRUE;
END_IF;

(* Main process logic - only active when system is running *)
IF SystemActive THEN
    (* Dough preparation phase *)
    IF NOT DoughReadySensor THEN
        DoughRollerMotor := TRUE;
        ToppingDispenser := FALSE;
        ConveyorMotor := FALSE;
        OvenHeater := FALSE;
        OvenTemperature := 0;
        BakingActive := FALSE;

    (* Topping application phase *)
    ELSIF DoughReadySensor AND NOT ToppingsReadySensor THEN
        DoughRollerMotor := FALSE;
        ToppingDispenser := TRUE;
        ConveyorMotor := FALSE;
        OvenHeater := FALSE;
        OvenTemperature := 0;
        BakingActive := FALSE;

    (* Baking phase - move to oven and bake *)
    ELSIF DoughReadySensor AND ToppingsReadySensor AND NOT BakingDoneSensor THEN
        DoughRollerMotor := FALSE;
        ToppingDispenser := FALSE;

        (* Conveyor runs until pizza is in oven, then oven heats *)
        IF NOT BakingActive THEN
            ConveyorMotor := TRUE;
            OvenHeater := FALSE;
            OvenTemperature := 0;
        ELSE
            ConveyorMotor := FALSE;
            OvenHeater := TRUE;
            OvenTemperature := 220;
        END_IF;

        (* Activate baking after conveyor has run *)
        BakingActive := TRUE;

    (* Baking complete - reset system *)
    ELSIF BakingDoneSensor AND BakingActive THEN
        DoughRollerMotor := FALSE;
        ToppingDispenser := FALSE;
        ConveyorMotor := FALSE;
        OvenHeater := FALSE;
        OvenTemperature := 0;
        BakingActive := FALSE;
        SystemActive := FALSE;

    (* Default safe state *)
    ELSE
        DoughRollerMotor := FALSE;
        ToppingDispenser := FALSE;
        ConveyorMotor := FALSE;
        OvenHeater := FALSE;
        OvenTemperature := 0;
        BakingActive := FALSE;
    END_IF;
ELSE
    (* System inactive - all outputs off *)
    DoughRollerMotor := FALSE;
    ToppingDispenser := FALSE;
    ConveyorMotor := FALSE;
    OvenHeater := FALSE;
    OvenTemperature := 0;
    BakingActive := FALSE;
END_IF;

END_FUNCTION_BLOCK;

(* ---- med_52.st ---- *)
FUNCTION_BLOCK TrafficManagementSystem
VAR_INPUT
    VehicleCount1 : INT;
    VehicleCount2 : INT;
    VehicleCount3 : INT;
    VehicleCount4 : INT;
END_VAR

VAR_OUTPUT
    TrafficLight1 : BOOL;
    TrafficLight2 : BOOL;
    TrafficLight3 : BOOL;
    TrafficLight4 : BOOL;
END_VAR

VAR
    (* No internal variables required for this logic *)
END_VAR

(* Main logic for intersection pair 1 and 2 *)
IF VehicleCount1 > VehicleCount2 THEN
    TrafficLight1 := TRUE;
    TrafficLight2 := FALSE;
ELSIF VehicleCount2 > VehicleCount1 THEN
    TrafficLight1 := FALSE;
    TrafficLight2 := TRUE;
ELSE
    (* Equal counts: default to intersection 1 green *)
    TrafficLight1 := TRUE;
    TrafficLight2 := FALSE;
END_IF;

(* Main logic for intersection pair 3 and 4 *)
IF VehicleCount3 > VehicleCount4 THEN
    TrafficLight3 := TRUE;
    TrafficLight4 := FALSE;
ELSIF VehicleCount4 > VehicleCount3 THEN
    TrafficLight3 := FALSE;
    TrafficLight4 := TRUE;
ELSE
    (* Equal counts: default to intersection 3 green *)
    TrafficLight3 := TRUE;
    TrafficLight4 := FALSE;
END_IF;

END_FUNCTION_BLOCK;

(* ---- med_53.st ---- *)
FUNCTION_BLOCK PouchMachine
VAR_INPUT
    start_machine: BOOL;
    stop_machine: BOOL;
END_VAR

VAR_OUTPUT
    machine_ready: BOOL;
    feeder_running: BOOL;
    cutter_running: BOOL;
    heating_running: BOOL;
    cooling_running: BOOL;
END_VAR

VAR
    startup_complete: BOOL := FALSE;
    shutdown_complete: BOOL := FALSE;
    state: INT := 0;
END_VAR

CASE state OF
    0:
        machine_ready := FALSE;
        feeder_running := FALSE;
        cutter_running := FALSE;
        heating_running := FALSE;
        cooling_running := FALSE;
        startup_complete := FALSE;
        shutdown_complete := FALSE;
        IF start_machine THEN
            state := 1;
        END_IF;
    1:
        heating_running := TRUE;
        state := 2;
    2:
        cooling_running := TRUE;
        state := 3;
    3:
        feeder_running := TRUE;
        state := 4;
    4:
        cutter_running := TRUE;
        state := 5;
    5:
        machine_ready := TRUE;
        startup_complete := TRUE;
        shutdown_complete := FALSE;
        IF stop_machine THEN
            state := 10;
        END_IF;
    10:
        cutter_running := FALSE;
        state := 11;
    11:
        feeder_running := FALSE;
        state := 12;
    12:
        cooling_running := FALSE;
        state := 13;
    13:
        heating_running := FALSE;
        state := 14;
    14:
        machine_ready := FALSE;
        startup_complete := FALSE;
        shutdown_complete := TRUE;
        state := 0;
    ELSE
        state := 0;
END_CASE;

END_FUNCTION_BLOCK;

(* ---- med_54.st ---- *)
FUNCTION_BLOCK FeedForwardControl
VAR_INPUT
    FlowRate1: REAL;
    FlowRate2: REAL;
    MixRatio: REAL;
END_VAR

VAR_OUTPUT
    OutFlowRate1: REAL;
    OutFlowRate2: REAL;
END_VAR

VAR
    MixedFlowRate: REAL;
    TempFlow1: REAL;
    TempFlow2: REAL;
END_VAR

(* Limit input flow rates to 0-100 range *)
IF FlowRate1 < 0.0 THEN
    TempFlow1 := 0.0;
ELSIF FlowRate1 > 100.0 THEN
    TempFlow1 := 100.0;
ELSE
    TempFlow1 := FlowRate1;
END_IF;

IF FlowRate2 < 0.0 THEN
    TempFlow2 := 0.0;
ELSIF FlowRate2 > 100.0 THEN
    TempFlow2 := 100.0;
ELSE
    TempFlow2 := FlowRate2;
END_IF;

(* Calculate total mixed flow rate *)
MixedFlowRate := TempFlow1 + TempFlow2;

(* Calculate output flow rates with division by zero protection *)
IF (MixRatio + 1.0) <> 0.0 AND MixedFlowRate <> 0.0 THEN
    OutFlowRate1 := MixedFlowRate * (MixRatio / (MixRatio + 1.0));
    OutFlowRate2 := MixedFlowRate * (1.0 / (MixRatio + 1.0));
ELSE
    OutFlowRate1 := 0.0;
    OutFlowRate2 := 0.0;
END_IF;

(* Limit output flow rates to 0-100 range *)
IF OutFlowRate1 < 0.0 THEN
    OutFlowRate1 := 0.0;
ELSIF OutFlowRate1 > 100.0 THEN
    OutFlowRate1 := 100.0;
END_IF;

IF OutFlowRate2 < 0.0 THEN
    OutFlowRate2 := 0.0;
ELSIF OutFlowRate2 > 100.0 THEN
    OutFlowRate2 := 100.0;
END_IF;

END_FUNCTION_BLOCK;

(* ---- med_55.st ---- *)
FUNCTION_BLOCK StateMachineControl
VAR_INPUT
    request : BOOL;
    done : BOOL;
END_VAR

VAR_OUTPUT
    listen : BOOL;
END_VAR

VAR
    state : INT := 0;
END_VAR

(* Main state machine logic *)
CASE state OF
    0: (* Idle state *)
        listen := TRUE;
        IF request THEN
            state := 1;
            listen := FALSE;
        END_IF;

    1: (* Processing state *)
        listen := FALSE;
        IF done THEN
            state := 0;
        END_IF;

    ELSE
        (* Safety fallback: reset to idle state *)
        state := 0;
        listen := TRUE;
END_CASE;

END_FUNCTION_BLOCK;

(* ---- med_56.st ---- *)
FUNCTION_BLOCK FB_SimpleRepeat
VAR_INPUT
    INPUT_VAR1 : INT := 2;
    INPUT_COUNTER : INT := 4;
END_VAR

VAR_OUTPUT
    OUTPUT_VAR1 : INT;
END_VAR

VAR
    COUNTER : INT;
END_VAR

OUTPUT_VAR1 := INPUT_VAR1;
COUNTER := INPUT_COUNTER;

IF COUNTER > 0 THEN
    REPEAT
        OUTPUT_VAR1 := OUTPUT_VAR1 * 2;
        COUNTER := COUNTER - 1;
    UNTIL COUNTER = 0
    END_REPEAT;
END_IF;

END_FUNCTION_BLOCK;

(* ---- med_57.st ---- *)
FUNCTION_BLOCK FB_CourseDifferenceControl
VAR_INPUT
    KOMPASS_GRAD : INT;
    KURS : INT;
END_VAR

VAR_OUTPUT
    KURS_DIFF : INT;
END_VAR

VAR
    iTempDiff : INT;
END_VAR

IF KOMPASS_GRAD < 0 THEN
    KURS_DIFF := 0;
ELSE
    iTempDiff := KURS - KOMPASS_GRAD;

    IF iTempDiff > 1800 THEN
        iTempDiff := iTempDiff - 3600;
    ELSIF iTempDiff < -1800 THEN
        iTempDiff := iTempDiff + 3600;
    END_IF;

    KURS_DIFF := iTempDiff;
END_IF;

END_FUNCTION_BLOCK

(* ---- med_58.st ---- *)
FUNCTION_BLOCK FB_ThresholdAccumulator
VAR_INPUT
    i : INT;
END_VAR

VAR_OUTPUT
    o : INT;
END_VAR

VAR
    s1 : INT;
END_VAR

s1 := 0;
IF i > 0 THEN
    s1 := s1 + i;
END_IF;
IF s1 = 42 THEN
    s1 := s1 + 8000;
END_IF;
IF s1 < 0 THEN
    o := 0;
ELSE
    o := s1;
END_IF;
END_FUNCTION_BLOCK

(* ---- med_59.st ---- *)
FUNCTION_BLOCK FB_ConditionalSelectAndAggregate
VAR_INPUT
Z : INT;
END_VAR

VAR_OUTPUT
NEW_Z : INT;
END_VAR

VAR
A_X : INT := 42;
A_Y : INT := 333;
END_VAR

IF A_X > Z THEN
    NEW_Z := A_Y;
ELSE
    NEW_Z := Z;
END_IF;
NEW_Z := NEW_Z + A_X + A_Y;
END_FUNCTION_BLOCK

(* ---- med_60.st ---- *)
FUNCTION_BLOCK FB_RequestHandler
    VAR_INPUT
        request : BOOL;
        done : BOOL;
    END_VAR

    VAR_OUTPUT
        listen : BOOL;
    END_VAR

    VAR
        state : INT := 0;
    END_VAR

    CASE state OF
        0:
            listen := TRUE;
            IF request THEN
                listen := FALSE;
                state := 1;
            END_IF;
        1:
            listen := FALSE;
            IF done THEN
                listen := TRUE;
                state := 0;
            END_IF;
    END_CASE;

END_FUNCTION_BLOCK;

(* ---- med_61.st ---- *)
FUNCTION_BLOCK FB_Sum
VAR_INPUT
    maxValue : INT;
END_VAR
VAR_OUTPUT
    wData : WORD;
END_VAR
VAR
    II : INT;
    tempSum : DINT;
END_VAR

tempSum := 0;
FOR II := 0 TO maxValue DO
    tempSum := tempSum + INT_TO_DINT(II);
END_FOR;
wData := DINT_TO_WORD(tempSum);
END_FUNCTION_BLOCK
